:SR[23]=$SCR_GRP[1].$MCH_POS_X;
:SR[24]=$SCR_GRP[1].$MCH_POS_Y;
2027: L P[2027] 800cm/min CNT100 COORD PTH ;
:SR[23]=$SCR_GRP[1].$MCH_POS_X;
:SR[24]=$SCR_GRP[1].$MCH_POS_Y;
2028: L P[2028] 800cm/min CNT100 COORD PTH ;
:SR[23]=$SCR_GRP[1].$MCH_POS_X;
:SR[24]=$SCR_GRP[1].$MCH_POS_Y;
2029: L P[2029] 800cm/min CNT100 COORD PTH ;
:SR[23]=$SCR_GRP[1].$MCH_POS_X;
:SR[24]=$SCR_GRP[1].$MCH_POS_Y;
2030: L P[2030] 800cm/min CNT100 COORD PTH ;
:SR[23]=$SCR_GRP[1].$MCH_POS_X;
:SR[24]=$SCR_GRP[1].$MCH_POS_Y;
2031: L P[2031] 800cm/min CNT100 COORD PTH ;
:SR[23]=$SCR_GRP[1].$MCH_POS_X;
:SR[24]=$SCR_GRP[1].$MCH_POS_Y;
2032: L P[2032] 800cm/min CNT100 COORD PTH ;
:SR[23]=$SCR_GRP[1].$MCH_POS_X;
:SR[24]=$SCR_GRP[1].$MCH_POS_Y;
2033: L P[2033] 800cm/min CNT100 COORD PTH ;
:SR[23]=$SCR_GRP[1].$MCH_POS_X;
:SR[24]=$SCR_GRP[1].$MCH_POS_Y;
2034: L P[2034] 800cm/min CNT100 COORD PTH ;
:SR[23]=$SCR_GRP[1].$MCH_POS_X;
:SR[24]=$SCR_GRP[1].$MCH_POS_Y;
2035: L P[2035] 800cm/min CNT100 COORD PTH ;
:SR[23]=$SCR_GRP[1].$MCH_POS_X;
:SR[24]=$SCR_GRP[1].$MCH_POS_Y;
2036: L P[2036] 800cm/min CNT100 COORD PTH ;
:SR[23]=$SCR_GRP[1].$MCH_POS_X;
:SR[24]=$SCR_GRP[1].$MCH_POS_Y;
2037: L P[2037] 800cm/min CNT100 COORD PTH ;
:SR[23]=$SCR_GRP[1].$MCH_POS_X;
:SR[24]=$SCR_GRP[1].$MCH_POS_Y;
2038: L P[2038] 800cm/min CNT100 COORD PTH ;
:SR[23]=$SCR_GRP[1].$MCH_POS_X;
:SR[24]=$SCR_GRP[1].$MCH_POS_Y;
2039: L P[2039] 800cm/min CNT100 COORD PTH ;
:SR[23]=$SCR_GRP[1].$MCH_POS_X;
:SR[24]=$SCR_GRP[1].$MCH_POS_Y;
2040: L P[2040] 800cm/min CNT100 COORD PTH ;
:SR[23]=$SCR_GRP[1].$MCH_POS_X;
:SR[24]=$SCR_GRP[1].$MCH_POS_Y;
2041: L P[2041] 800cm/min CNT100 COORD PTH ;
:SR[23]=$SCR_GRP[1].$MCH_POS_X;
:SR[24]=$SCR_GRP[1].$MCH_POS_Y;
2042: L P[2042] 800cm/min CNT100 COORD PTH ;
:SR[23]=$SCR_GRP[1].$MCH_POS_X;
:SR[24]=$SCR_GRP[1].$MCH_POS_Y;
2043: L P[2043] 800cm/min CNT100 COORD PTH ;
:SR[23]=$SCR_GRP[1].$MCH_POS_X;
:SR[24]=$SCR_GRP[1].$MCH_POS_Y;
2044: L P[2044] 800cm/min CNT100 COORD PTH ;
:SR[23]=$SCR_GRP[1].$MCH_POS_X;
:SR[24]=$SCR_GRP[1].$MCH_POS_Y;
2045: L P[2045] 800cm/min CNT100 COORD PTH ;
:SR[23]=$SCR_GRP[1].$MCH_POS_X;
:SR[24]=$SCR_GRP[1].$MCH_POS_Y;
2046: L P[2046] 800cm/min CNT100 COORD PTH ;
:SR[23]=$SCR_GRP[1].$MCH_POS_X;
:SR[24]=$SCR_GRP[1].$MCH_POS_Y;
2047: L P[2047] 800cm/min CNT100 COORD PTH ;
:SR[23]=$SCR_GRP[1].$MCH_POS_X;
:SR[24]=$SCR_GRP[1].$MCH_POS_Y;
2048: L P[2048] 800cm/min CNT100 COORD PTH ;
:SR[23]=$SCR_GRP[1].$MCH_POS_X;
:SR[24]=$SCR_GRP[1].$MCH_POS_Y;
2049: L P[2049] 800cm/min CNT100 COORD PTH ;
:SR[23]=$SCR_GRP[1].$MCH_POS_X;
:SR[24]=$SCR_GRP[1].$MCH_POS_Y;
2050: L P[2050] 800cm/min CNT100 COORD PTH ;
:SR[23]=$SCR_GRP[1].$MCH_POS_X;
:SR[24]=$SCR_GRP[1].$MCH_POS_Y;
2051: L P[2051] 800cm/min CNT100 COORD PTH ;
:SR[23]=$SCR_GRP[1].$MCH_POS_X;
:SR[24]=$SCR_GRP[1].$MCH_POS_Y;
2052: L P[2052] 800cm/min CNT100 COORD PTH ;
:SR[23]=$SCR_GRP[1].$MCH_POS_X;
:SR[24]=$SCR_GRP[1].$MCH_POS_Y;
2053: L P[2053] 800cm/min CNT100 COORD PTH ;
:SR[23]=$SCR_GRP[1].$MCH_POS_X;
:SR[24]=$SCR_GRP[1].$MCH_POS_Y;
2054: L P[2054] 800cm/min CNT100 COORD PTH ;
:SR[23]=$SCR_GRP[1].$MCH_POS_X;
:SR[24]=$SCR_GRP[1].$MCH_POS_Y;
2055: L P[2055] 800cm/min CNT100 COORD PTH ;
:SR[23]=$SCR_GRP[1].$MCH_POS_X;
:SR[24]=$SCR_GRP[1].$MCH_POS_Y;
2056: L P[2056] 800cm/min CNT100 COORD PTH ;
:SR[23]=$SCR_GRP[1].$MCH_POS_X;
:SR[24]=$SCR_GRP[1].$MCH_POS_Y;
2057: L P[2057] 800cm/min CNT100 COORD PTH ;
:SR[23]=$SCR_GRP[1].$MCH_POS_X;
:SR[24]=$SCR_GRP[1].$MCH_POS_Y;
2058: L P[2058] 800cm/min CNT100 COORD PTH ;
:SR[23]=$SCR_GRP[1].$MCH_POS_X;
:SR[24]=$SCR_GRP[1].$MCH_POS_Y;
2059: L P[2059] 800cm/min CNT100 COORD PTH ;
:SR[23]=$SCR_GRP[1].$MCH_POS_X;
:SR[24]=$SCR_GRP[1].$MCH_POS_Y;
2060: L P[2060] 800cm/min CNT100 COORD PTH ;
:SR[23]=$SCR_GRP[1].$MCH_POS_X;
:SR[24]=$SCR_GRP[1].$MCH_POS_Y;
2061: L P[2061] 800cm/min CNT100 COORD PTH ;
:SR[23]=$SCR_GRP[1].$MCH_POS_X;
:SR[24]=$SCR_GRP[1].$MCH_POS_Y;
2062: L P[2062] 800cm/min CNT100 COORD PTH ;
:SR[23]=$SCR_GRP[1].$MCH_POS_X;
:SR[24]=$SCR_GRP[1].$MCH_POS_Y;
2063: L P[2063] 800cm/min CNT100 COORD PTH ;
:SR[23]=$SCR_GRP[1].$MCH_POS_X;
:SR[24]=$SCR_GRP[1].$MCH_POS_Y;
2064: L P[2064] 800cm/min CNT100 COORD PTH ;
:SR[23]=$SCR_GRP[1].$MCH_POS_X;
:SR[24]=$SCR_GRP[1].$MCH_POS_Y;
2065: L P[2065] 800cm/min CNT100 COORD PTH ;
:SR[23]=$SCR_GRP[1].$MCH_POS_X;
:SR[24]=$SCR_GRP[1].$MCH_POS_Y;
2066: L P[2066] 800cm/min CNT100 COORD PTH ;
:SR[23]=$SCR_GRP[1].$MCH_POS_X;
:SR[24]=$SCR_GRP[1].$MCH_POS_Y;
2067: L P[2067] 800cm/min CNT100 COORD PTH ;
:SR[23]=$SCR_GRP[1].$MCH_POS_X;
:SR[24]=$SCR_GRP[1].$MCH_POS_Y;
2068: L P[2068] 800cm/min CNT100 COORD PTH ;
:SR[23]=$SCR_GRP[1].$MCH_POS_X;
:SR[24]=$SCR_GRP[1].$MCH_POS_Y;
2069: L P[2069] 800cm/min CNT100 COORD PTH ;
:SR[23]=$SCR_GRP[1].$MCH_POS_X;
:SR[24]=$SCR_GRP[1].$MCH_POS_Y;
2070: L P[2070] 800cm/min CNT100 COORD PTH ;
:SR[23]=$SCR_GRP[1].$MCH_POS_X;
:SR[24]=$SCR_GRP[1].$MCH_POS_Y;
2071: L P[2071] 800cm/min CNT100 COORD PTH ;
:SR[23]=$SCR_GRP[1].$MCH_POS_X;
:SR[24]=$SCR_GRP[1].$MCH_POS_Y;
2072: L P[2072] 800cm/min CNT100 COORD PTH ;
:SR[23]=$SCR_GRP[1].$MCH_POS_X;
:SR[24]=$SCR_GRP[1].$MCH_POS_Y;
2073: L P[2073] 800cm/min CNT100 COORD PTH ;
:SR[23]=$SCR_GRP[1].$MCH_POS_X;
:SR[24]=$SCR_GRP[1].$MCH_POS_Y;
2074: L P[2074] 800cm/min CNT100 COORD PTH ;
:SR[23]=$SCR_GRP[1].$MCH_POS_X;
:SR[24]=$SCR_GRP[1].$MCH_POS_Y;
2075: L P[2075] 800cm/min CNT100 COORD PTH ;
:SR[23]=$SCR_GRP[1].$MCH_POS_X;
:SR[24]=$SCR_GRP[1].$MCH_POS_Y;
2076: L P[2076] 800cm/min CNT100 COORD PTH ;
:SR[23]=$SCR_GRP[1].$MCH_POS_X;
:SR[24]=$SCR_GRP[1].$MCH_POS_Y;
2077: L P[2077] 800cm/min CNT100 COORD PTH ;
:SR[23]=$SCR_GRP[1].$MCH_POS_X;
:SR[24]=$SCR_GRP[1].$MCH_POS_Y;
2078: L P[2078] 800cm/min CNT100 COORD PTH ;
:SR[23]=$SCR_GRP[1].$MCH_POS_X;
:SR[24]=$SCR_GRP[1].$MCH_POS_Y;
2079: L P[2079] 800cm/min CNT100 COORD PTH ;
:SR[23]=$SCR_GRP[1].$MCH_POS_X;
:SR[24]=$SCR_GRP[1].$MCH_POS_Y;
2080: L P[2080] 800cm/min CNT100 COORD PTH ;
:SR[23]=$SCR_GRP[1].$MCH_POS_X;
:SR[24]=$SCR_GRP[1].$MCH_POS_Y;
2081: L P[2081] 800cm/min CNT100 COORD PTH ;
:SR[23]=$SCR_GRP[1].$MCH_POS_X;
:SR[24]=$SCR_GRP[1].$MCH_POS_Y;
2082: L P[2082] 800cm/min CNT100 COORD PTH ;
:SR[23]=$SCR_GRP[1].$MCH_POS_X;
:SR[24]=$SCR_GRP[1].$MCH_POS_Y;
2083: L P[2083] 800cm/min CNT100 COORD PTH ;
:SR[23]=$SCR_GRP[1].$MCH_POS_X;
:SR[24]=$SCR_GRP[1].$MCH_POS_Y;
2084: L P[2084] 800cm/min CNT100 COORD PTH ;
:SR[23]=$SCR_GRP[1].$MCH_POS_X;
:SR[24]=$SCR_GRP[1].$MCH_POS_Y;
2085: L P[2085] 800cm/min CNT100 COORD PTH ;
:SR[23]=$SCR_GRP[1].$MCH_POS_X;
:SR[24]=$SCR_GRP[1].$MCH_POS_Y;
2086: L P[2086] 800cm/min CNT100 COORD PTH ;
:SR[23]=$SCR_GRP[1].$MCH_POS_X;
:SR[24]=$SCR_GRP[1].$MCH_POS_Y;
2087: L P[2087] 800cm/min CNT100 COORD PTH ;
:SR[23]=$SCR_GRP[1].$MCH_POS_X;
:SR[24]=$SCR_GRP[1].$MCH_POS_Y;
2088: L P[2088] 800cm/min CNT100 COORD PTH ;
:SR[23]=$SCR_GRP[1].$MCH_POS_X;
:SR[24]=$SCR_GRP[1].$MCH_POS_Y;
2089: L P[2089] 800cm/min CNT100 COORD PTH ;
:SR[23]=$SCR_GRP[1].$MCH_POS_X;
:SR[24]=$SCR_GRP[1].$MCH_POS_Y;
2090: L P[2090] 800cm/min CNT100 COORD PTH ;
:SR[23]=$SCR_GRP[1].$MCH_POS_X;
:SR[24]=$SCR_GRP[1].$MCH_POS_Y;
2091: L P[2091] 800cm/min CNT100 COORD PTH ;
:SR[23]=$SCR_GRP[1].$MCH_POS_X;
:SR[24]=$SCR_GRP[1].$MCH_POS_Y;
2092: L P[2092] 800cm/min CNT100 COORD PTH ;
:SR[23]=$SCR_GRP[1].$MCH_POS_X;
:SR[24]=$SCR_GRP[1].$MCH_POS_Y;
2093: L P[2093] 800cm/min CNT100 COORD PTH ;
:SR[23]=$SCR_GRP[1].$MCH_POS_X;
:SR[24]=$SCR_GRP[1].$MCH_POS_Y;
2094: L P[2094] 800cm/min CNT100 COORD PTH ;
:SR[23]=$SCR_GRP[1].$MCH_POS_X;
:SR[24]=$SCR_GRP[1].$MCH_POS_Y;
2095: L P[2095] 800cm/min CNT100 COORD PTH ;
:SR[23]=$SCR_GRP[1].$MCH_POS_X;
:SR[24]=$SCR_GRP[1].$MCH_POS_Y;
2096: L P[2096] 800cm/min CNT100 COORD PTH ;
:SR[23]=$SCR_GRP[1].$MCH_POS_X;
:SR[24]=$SCR_GRP[1].$MCH_POS_Y;
2097: L P[2097] 800cm/min CNT100 COORD PTH ;
:SR[23]=$SCR_GRP[1].$MCH_POS_X;
:SR[24]=$SCR_GRP[1].$MCH_POS_Y;
2098: L P[2098] 800cm/min CNT100 COORD PTH ;
:SR[23]=$SCR_GRP[1].$MCH_POS_X;
:SR[24]=$SCR_GRP[1].$MCH_POS_Y;
2099: L P[2099] 800cm/min CNT100 COORD PTH ;
:SR[23]=$SCR_GRP[1].$MCH_POS_X;
:SR[24]=$SCR_GRP[1].$MCH_POS_Y;
2100: L P[2100] 800cm/min CNT100 COORD PTH ;
:SR[23]=$SCR_GRP[1].$MCH_POS_X;
:SR[24]=$SCR_GRP[1].$MCH_POS_Y;
2101: L P[2101] 800cm/min CNT100 COORD PTH ;
:SR[23]=$SCR_GRP[1].$MCH_POS_X;
:SR[24]=$SCR_GRP[1].$MCH_POS_Y;
2102: L P[2102] 800cm/min CNT100 COORD PTH ;
:SR[23]=$SCR_GRP[1].$MCH_POS_X;
:SR[24]=$SCR_GRP[1].$MCH_POS_Y;
2103: L P[2103] 800cm/min CNT100 COORD PTH ;
:SR[23]=$SCR_GRP[1].$MCH_POS_X;
:SR[24]=$SCR_GRP[1].$MCH_POS_Y;
2104: L P[2104] 800cm/min CNT100 COORD PTH ;
:SR[23]=$SCR_GRP[1].$MCH_POS_X;
:SR[24]=$SCR_GRP[1].$MCH_POS_Y;
2105: L P[2105] 800cm/min CNT100 COORD PTH ;
:SR[23]=$SCR_GRP[1].$MCH_POS_X;
:SR[24]=$SCR_GRP[1].$MCH_POS_Y;
2106: L P[2106] 800cm/min CNT100 COORD PTH ;
:SR[23]=$SCR_GRP[1].$MCH_POS_X;
:SR[24]=$SCR_GRP[1].$MCH_POS_Y;
2107: L P[2107] 800cm/min CNT100 COORD PTH ;
:SR[23]=$SCR_GRP[1].$MCH_POS_X;
:SR[24]=$SCR_GRP[1].$MCH_POS_Y;
2108: L P[2108] 800cm/min CNT100 COORD PTH ;
:SR[23]=$SCR_GRP[1].$MCH_POS_X;
:SR[24]=$SCR_GRP[1].$MCH_POS_Y;
2109: L P[2109] 800cm/min CNT100 COORD PTH ;
:SR[23]=$SCR_GRP[1].$MCH_POS_X;
:SR[24]=$SCR_GRP[1].$MCH_POS_Y;
2110: L P[2110] 800cm/min CNT100 COORD PTH ;
:SR[23]=$SCR_GRP[1].$MCH_POS_X;
:SR[24]=$SCR_GRP[1].$MCH_POS_Y;
2111: L P[2111] 800cm/min CNT100 COORD PTH ;
:SR[23]=$SCR_GRP[1].$MCH_POS_X;
:SR[24]=$SCR_GRP[1].$MCH_POS_Y;
2112: L P[2112] 800cm/min CNT100 COORD PTH ;
:SR[23]=$SCR_GRP[1].$MCH_POS_X;
:SR[24]=$SCR_GRP[1].$MCH_POS_Y;
2113: L P[2113] 800cm/min CNT100 COORD PTH ;
:SR[23]=$SCR_GRP[1].$MCH_POS_X;
:SR[24]=$SCR_GRP[1].$MCH_POS_Y;
2114: L P[2114] 800cm/min CNT100 COORD PTH ;
:SR[23]=$SCR_GRP[1].$MCH_POS_X;
:SR[24]=$SCR_GRP[1].$MCH_POS_Y;
2115: L P[2115] 800cm/min CNT100 COORD PTH ;
:SR[23]=$SCR_GRP[1].$MCH_POS_X;
:SR[24]=$SCR_GRP[1].$MCH_POS_Y;
2116: L P[2116] 800cm/min CNT100 COORD PTH ;
:SR[23]=$SCR_GRP[1].$MCH_POS_X;
:SR[24]=$SCR_GRP[1].$MCH_POS_Y;
2117: L P[2117] 800cm/min CNT100 COORD PTH ;
:SR[23]=$SCR_GRP[1].$MCH_POS_X;
:SR[24]=$SCR_GRP[1].$MCH_POS_Y;
2118: L P[2118] 800cm/min CNT100 COORD PTH ;
:SR[23]=$SCR_GRP[1].$MCH_POS_X;
:SR[24]=$SCR_GRP[1].$MCH_POS_Y;
2119: L P[2119] 800cm/min CNT100 COORD PTH ;
:SR[23]=$SCR_GRP[1].$MCH_POS_X;
:SR[24]=$SCR_GRP[1].$MCH_POS_Y;
2120: L P[2120] 800cm/min CNT100 COORD PTH ;
:SR[23]=$SCR_GRP[1].$MCH_POS_X;
:SR[24]=$SCR_GRP[1].$MCH_POS_Y;
2121: L P[2121] 800cm/min CNT100 COORD PTH ;
:SR[23]=$SCR_GRP[1].$MCH_POS_X;
:SR[24]=$SCR_GRP[1].$MCH_POS_Y;
2122: L P[2122] 800cm/min CNT100 COORD PTH ;
:SR[23]=$SCR_GRP[1].$MCH_POS_X;
:SR[24]=$SCR_GRP[1].$MCH_POS_Y;
2123: L P[2123] 800cm/min CNT100 COORD PTH ;
:SR[23]=$SCR_GRP[1].$MCH_POS_X;
:SR[24]=$SCR_GRP[1].$MCH_POS_Y;
2124: L P[2124] 800cm/min CNT100 COORD PTH ;
:SR[23]=$SCR_GRP[1].$MCH_POS_X;
:SR[24]=$SCR_GRP[1].$MCH_POS_Y;
2125: L P[2125] 800cm/min CNT100 COORD PTH ;
:SR[23]=$SCR_GRP[1].$MCH_POS_X;
:SR[24]=$SCR_GRP[1].$MCH_POS_Y;
2126: L P[2126] 800cm/min CNT100 COORD PTH ;
:SR[23]=$SCR_GRP[1].$MCH_POS_X;
:SR[24]=$SCR_GRP[1].$MCH_POS_Y;
2127: L P[2127] 800cm/min CNT100 COORD PTH ;
:SR[23]=$SCR_GRP[1].$MCH_POS_X;
:SR[24]=$SCR_GRP[1].$MCH_POS_Y;
2128: L P[2128] 800cm/min CNT100 COORD PTH ;
:SR[23]=$SCR_GRP[1].$MCH_POS_X;
:SR[24]=$SCR_GRP[1].$MCH_POS_Y;
2129: L P[2129] 800cm/min CNT100 COORD PTH ;
:SR[23]=$SCR_GRP[1].$MCH_POS_X;
:SR[24]=$SCR_GRP[1].$MCH_POS_Y;
2130: L P[2130] 800cm/min CNT100 COORD PTH ;
:SR[23]=$SCR_GRP[1].$MCH_POS_X;
:SR[24]=$SCR_GRP[1].$MCH_POS_Y;
2131: L P[2131] 800cm/min CNT100 COORD PTH ;
:SR[23]=$SCR_GRP[1].$MCH_POS_X;
:SR[24]=$SCR_GRP[1].$MCH_POS_Y;
2132: L P[2132] 800cm/min CNT100 COORD PTH ;
:SR[23]=$SCR_GRP[1].$MCH_POS_X;
:SR[24]=$SCR_GRP[1].$MCH_POS_Y;
2133: L P[2133] 800cm/min CNT100 COORD PTH ;
:SR[23]=$SCR_GRP[1].$MCH_POS_X;
:SR[24]=$SCR_GRP[1].$MCH_POS_Y;
2134: L P[2134] 800cm/min CNT100 COORD PTH ;
:SR[23]=$SCR_GRP[1].$MCH_POS_X;
:SR[24]=$SCR_GRP[1].$MCH_POS_Y;
2135: L P[2135] 800cm/min CNT100 COORD PTH ;
:SR[23]=$SCR_GRP[1].$MCH_POS_X;
:SR[24]=$SCR_GRP[1].$MCH_POS_Y;
2136: L P[2136] 800cm/min CNT100 COORD PTH ;
:SR[23]=$SCR_GRP[1].$MCH_POS_X;
:SR[24]=$SCR_GRP[1].$MCH_POS_Y;
2137: L P[2137] 800cm/min CNT100 COORD PTH ;
:SR[23]=$SCR_GRP[1].$MCH_POS_X;
:SR[24]=$SCR_GRP[1].$MCH_POS_Y;
2138: L P[2138] 800cm/min CNT100 COORD PTH ;
:SR[23]=$SCR_GRP[1].$MCH_POS_X;
:SR[24]=$SCR_GRP[1].$MCH_POS_Y;
2139: L P[2139] 800cm/min CNT100 COORD PTH ;
:SR[23]=$SCR_GRP[1].$MCH_POS_X;
:SR[24]=$SCR_GRP[1].$MCH_POS_Y;
2140: L P[2140] 800cm/min CNT100 COORD PTH ;
:SR[23]=$SCR_GRP[1].$MCH_POS_X;
:SR[24]=$SCR_GRP[1].$MCH_POS_Y;
2141: L P[2141] 800cm/min CNT100 COORD PTH ;
:SR[23]=$SCR_GRP[1].$MCH_POS_X;
:SR[24]=$SCR_GRP[1].$MCH_POS_Y;
2142: L P[2142] 800cm/min CNT100 COORD PTH ;
:SR[23]=$SCR_GRP[1].$MCH_POS_X;
:SR[24]=$SCR_GRP[1].$MCH_POS_Y;
2143: L P[2143] 800cm/min CNT100 COORD PTH ;
:SR[23]=$SCR_GRP[1].$MCH_POS_X;
:SR[24]=$SCR_GRP[1].$MCH_POS_Y;
2144: L P[2144] 800cm/min CNT100 COORD PTH ;
:SR[23]=$SCR_GRP[1].$MCH_POS_X;
:SR[24]=$SCR_GRP[1].$MCH_POS_Y;
2145: L P[2145] 800cm/min CNT100 COORD PTH ;
:SR[23]=$SCR_GRP[1].$MCH_POS_X;
:SR[24]=$SCR_GRP[1].$MCH_POS_Y;
2146: L P[2146] 800cm/min CNT100 COORD PTH ;
:SR[23]=$SCR_GRP[1].$MCH_POS_X;
:SR[24]=$SCR_GRP[1].$MCH_POS_Y;
2147: L P[2147] 800cm/min CNT100 COORD PTH ;
:SR[23]=$SCR_GRP[1].$MCH_POS_X;
:SR[24]=$SCR_GRP[1].$MCH_POS_Y;
2148: L P[2148] 800cm/min CNT100 COORD PTH ;
:SR[23]=$SCR_GRP[1].$MCH_POS_X;
:SR[24]=$SCR_GRP[1].$MCH_POS_Y;
2149: L P[2149] 800cm/min CNT100 COORD PTH ;
:SR[23]=$SCR_GRP[1].$MCH_POS_X;
:SR[24]=$SCR_GRP[1].$MCH_POS_Y;
2150: L P[2150] 800cm/min CNT100 COORD PTH ;
:SR[23]=$SCR_GRP[1].$MCH_POS_X;
:SR[24]=$SCR_GRP[1].$MCH_POS_Y;
2151: L P[2151] 800cm/min CNT100 COORD PTH ;
:SR[23]=$SCR_GRP[1].$MCH_POS_X;
:SR[24]=$SCR_GRP[1].$MCH_POS_Y;
2152: L P[2152] 800cm/min CNT100 COORD PTH ;
:SR[23]=$SCR_GRP[1].$MCH_POS_X;
:SR[24]=$SCR_GRP[1].$MCH_POS_Y;
2153: L P[2153] 800cm/min CNT100 COORD PTH ;
:SR[23]=$SCR_GRP[1].$MCH_POS_X;
:SR[24]=$SCR_GRP[1].$MCH_POS_Y;
2154: L P[2154] 800cm/min CNT100 COORD PTH ;
:SR[23]=$SCR_GRP[1].$MCH_POS_X;
:SR[24]=$SCR_GRP[1].$MCH_POS_Y;
2155: L P[2155] 800cm/min CNT100 COORD PTH ;
:SR[23]=$SCR_GRP[1].$MCH_POS_X;
:SR[24]=$SCR_GRP[1].$MCH_POS_Y;
2156: L P[2156] 800cm/min CNT100 COORD PTH ;
:SR[23]=$SCR_GRP[1].$MCH_POS_X;
:SR[24]=$SCR_GRP[1].$MCH_POS_Y;
2157: L P[2157] 800cm/min CNT100 COORD PTH ;
:SR[23]=$SCR_GRP[1].$MCH_POS_X;
:SR[24]=$SCR_GRP[1].$MCH_POS_Y;
2158: L P[2158] 800cm/min CNT100 COORD PTH ;
:SR[23]=$SCR_GRP[1].$MCH_POS_X;
:SR[24]=$SCR_GRP[1].$MCH_POS_Y;
2159: L P[2159] 800cm/min CNT100 COORD PTH ;
:SR[23]=$SCR_GRP[1].$MCH_POS_X;
:SR[24]=$SCR_GRP[1].$MCH_POS_Y;
2160: L P[2160] 800cm/min CNT100 COORD PTH ;
:SR[23]=$SCR_GRP[1].$MCH_POS_X;
:SR[24]=$SCR_GRP[1].$MCH_POS_Y;
2161: L P[2161] 800cm/min CNT100 COORD PTH ;
:SR[23]=$SCR_GRP[1].$MCH_POS_X;
:SR[24]=$SCR_GRP[1].$MCH_POS_Y;
2162: L P[2162] 800cm/min CNT100 COORD PTH ;
:SR[23]=$SCR_GRP[1].$MCH_POS_X;
:SR[24]=$SCR_GRP[1].$MCH_POS_Y;
2163: L P[2163] 800cm/min CNT100 COORD PTH ;
:SR[23]=$SCR_GRP[1].$MCH_POS_X;
:SR[24]=$SCR_GRP[1].$MCH_POS_Y;
2164: L P[2164] 800cm/min CNT100 COORD PTH ;
:SR[23]=$SCR_GRP[1].$MCH_POS_X;
:SR[24]=$SCR_GRP[1].$MCH_POS_Y;
2165: L P[2165] 800cm/min CNT100 COORD PTH ;
:SR[23]=$SCR_GRP[1].$MCH_POS_X;
:SR[24]=$SCR_GRP[1].$MCH_POS_Y;
2166: L P[2166] 800cm/min CNT100 COORD PTH ;
:SR[23]=$SCR_GRP[1].$MCH_POS_X;
:SR[24]=$SCR_GRP[1].$MCH_POS_Y;
2167: L P[2167] 800cm/min CNT100 COORD PTH ;
:SR[23]=$SCR_GRP[1].$MCH_POS_X;
:SR[24]=$SCR_GRP[1].$MCH_POS_Y;
2168: L P[2168] 800cm/min CNT100 COORD PTH ;
:SR[23]=$SCR_GRP[1].$MCH_POS_X;
:SR[24]=$SCR_GRP[1].$MCH_POS_Y;
2169: L P[2169] 800cm/min CNT100 COORD PTH ;
:SR[23]=$SCR_GRP[1].$MCH_POS_X;
:SR[24]=$SCR_GRP[1].$MCH_POS_Y;
2170: L P[2170] 800cm/min CNT100 COORD PTH ;
:SR[23]=$SCR_GRP[1].$MCH_POS_X;
:SR[24]=$SCR_GRP[1].$MCH_POS_Y;
2171: L P[2171] 800cm/min CNT100 COORD PTH ;
:SR[23]=$SCR_GRP[1].$MCH_POS_X;
:SR[24]=$SCR_GRP[1].$MCH_POS_Y;
2172: L P[2172] 800cm/min CNT100 COORD PTH ;
:SR[23]=$SCR_GRP[1].$MCH_POS_X;
:SR[24]=$SCR_GRP[1].$MCH_POS_Y;
2173: L P[2173] 800cm/min CNT100 COORD PTH ;
:SR[23]=$SCR_GRP[1].$MCH_POS_X;
:SR[24]=$SCR_GRP[1].$MCH_POS_Y;
2174: L P[2174] 800cm/min CNT100 COORD PTH ;
:SR[23]=$SCR_GRP[1].$MCH_POS_X;
:SR[24]=$SCR_GRP[1].$MCH_POS_Y;
2175: L P[2175] 800cm/min CNT100 COORD PTH ;
:SR[23]=$SCR_GRP[1].$MCH_POS_X;
:SR[24]=$SCR_GRP[1].$MCH_POS_Y;
2176: L P[2176] 800cm/min CNT100 COORD PTH ;
:SR[23]=$SCR_GRP[1].$MCH_POS_X;
:SR[24]=$SCR_GRP[1].$MCH_POS_Y;
2177: L P[2177] 800cm/min CNT100 COORD PTH ;
:SR[23]=$SCR_GRP[1].$MCH_POS_X;
:SR[24]=$SCR_GRP[1].$MCH_POS_Y;
2178: L P[2178] 800cm/min CNT100 COORD PTH ;
:SR[23]=$SCR_GRP[1].$MCH_POS_X;
:SR[24]=$SCR_GRP[1].$MCH_POS_Y;
2179: L P[2179] 800cm/min CNT100 COORD PTH ;
:SR[23]=$SCR_GRP[1].$MCH_POS_X;
:SR[24]=$SCR_GRP[1].$MCH_POS_Y;
2180: L P[2180] 800cm/min CNT100 COORD PTH ;
:SR[23]=$SCR_GRP[1].$MCH_POS_X;
:SR[24]=$SCR_GRP[1].$MCH_POS_Y;
2181: L P[2181] 800cm/min CNT100 COORD PTH ;
:SR[23]=$SCR_GRP[1].$MCH_POS_X;
:SR[24]=$SCR_GRP[1].$MCH_POS_Y;
2182: L P[2182] 800cm/min CNT100 COORD PTH ;
:SR[23]=$SCR_GRP[1].$MCH_POS_X;
:SR[24]=$SCR_GRP[1].$MCH_POS_Y;
2183: L P[2183] 800cm/min CNT100 COORD PTH ;
:SR[23]=$SCR_GRP[1].$MCH_POS_X;
:SR[24]=$SCR_GRP[1].$MCH_POS_Y;
2184: L P[2184] 800cm/min CNT100 COORD PTH ;
:SR[23]=$SCR_GRP[1].$MCH_POS_X;
:SR[24]=$SCR_GRP[1].$MCH_POS_Y;
2185: L P[2185] 800cm/min CNT100 COORD PTH ;
:SR[23]=$SCR_GRP[1].$MCH_POS_X;
:SR[24]=$SCR_GRP[1].$MCH_POS_Y;
2186: L P[2186] 800cm/min CNT100 COORD PTH ;
:SR[23]=$SCR_GRP[1].$MCH_POS_X;
:SR[24]=$SCR_GRP[1].$MCH_POS_Y;
2187: L P[2187] 800cm/min CNT100 COORD PTH ;
:SR[23]=$SCR_GRP[1].$MCH_POS_X;
:SR[24]=$SCR_GRP[1].$MCH_POS_Y;
2188: L P[2188] 800cm/min CNT100 COORD PTH ;
:SR[23]=$SCR_GRP[1].$MCH_POS_X;
:SR[24]=$SCR_GRP[1].$MCH_POS_Y;
2189: L P[2189] 800cm/min CNT100 COORD PTH ;
:SR[23]=$SCR_GRP[1].$MCH_POS_X;
:SR[24]=$SCR_GRP[1].$MCH_POS_Y;
2190: L P[2190] 800cm/min CNT100 COORD PTH ;
:SR[23]=$SCR_GRP[1].$MCH_POS_X;
:SR[24]=$SCR_GRP[1].$MCH_POS_Y;
2191: L P[2191] 800cm/min CNT100 COORD PTH ;
:SR[23]=$SCR_GRP[1].$MCH_POS_X;
:SR[24]=$SCR_GRP[1].$MCH_POS_Y;
2192: L P[2192] 800cm/min CNT100 COORD PTH ;
:SR[23]=$SCR_GRP[1].$MCH_POS_X;
:SR[24]=$SCR_GRP[1].$MCH_POS_Y;
2193: L P[2193] 800cm/min CNT100 COORD PTH ;
:SR[23]=$SCR_GRP[1].$MCH_POS_X;
:SR[24]=$SCR_GRP[1].$MCH_POS_Y;
2194: L P[2194] 800cm/min CNT100 COORD PTH ;
:SR[23]=$SCR_GRP[1].$MCH_POS_X;
:SR[24]=$SCR_GRP[1].$MCH_POS_Y;
2195: L P[2195] 800cm/min CNT100 COORD PTH ;
:SR[23]=$SCR_GRP[1].$MCH_POS_X;
:SR[24]=$SCR_GRP[1].$MCH_POS_Y;
2196: L P[2196] 800cm/min CNT100 COORD PTH ;
:SR[23]=$SCR_GRP[1].$MCH_POS_X;
:SR[24]=$SCR_GRP[1].$MCH_POS_Y;
2197: L P[2197] 800cm/min CNT100 COORD PTH ;
:SR[23]=$SCR_GRP[1].$MCH_POS_X;
:SR[24]=$SCR_GRP[1].$MCH_POS_Y;
2198: L P[2198] 800cm/min CNT100 COORD PTH ;
:SR[23]=$SCR_GRP[1].$MCH_POS_X;
:SR[24]=$SCR_GRP[1].$MCH_POS_Y;
2199: L P[2199] 800cm/min CNT100 COORD PTH ;
:SR[23]=$SCR_GRP[1].$MCH_POS_X;
:SR[24]=$SCR_GRP[1].$MCH_POS_Y;
2200: L P[2200] 800cm/min CNT100 COORD PTH ;
:SR[23]=$SCR_GRP[1].$MCH_POS_X;
:SR[24]=$SCR_GRP[1].$MCH_POS_Y;
2201: L P[2201] 800cm/min CNT100 COORD PTH ;
:SR[23]=$SCR_GRP[1].$MCH_POS_X;
:SR[24]=$SCR_GRP[1].$MCH_POS_Y;
2202: L P[2202] 800cm/min CNT100 COORD PTH ;
:SR[23]=$SCR_GRP[1].$MCH_POS_X;
:SR[24]=$SCR_GRP[1].$MCH_POS_Y;
2203: L P[2203] 800cm/min CNT100 COORD PTH ;
:SR[23]=$SCR_GRP[1].$MCH_POS_X;
:SR[24]=$SCR_GRP[1].$MCH_POS_Y;
2204: L P[2204] 800cm/min CNT100 COORD PTH ;
:SR[23]=$SCR_GRP[1].$MCH_POS_X;
:SR[24]=$SCR_GRP[1].$MCH_POS_Y;
2205: L P[2205] 800cm/min CNT100 COORD PTH ;
:SR[23]=$SCR_GRP[1].$MCH_POS_X;
:SR[24]=$SCR_GRP[1].$MCH_POS_Y;
2206: L P[2206] 800cm/min CNT100 COORD PTH ;
:SR[23]=$SCR_GRP[1].$MCH_POS_X;
:SR[24]=$SCR_GRP[1].$MCH_POS_Y;
2207: L P[2207] 800cm/min CNT100 COORD PTH ;
:SR[23]=$SCR_GRP[1].$MCH_POS_X;
:SR[24]=$SCR_GRP[1].$MCH_POS_Y;
2208: L P[2208] 800cm/min CNT100 COORD PTH ;
:SR[23]=$SCR_GRP[1].$MCH_POS_X;
:SR[24]=$SCR_GRP[1].$MCH_POS_Y;
2209: L P[2209] 800cm/min CNT100 COORD PTH ;
:SR[23]=$SCR_GRP[1].$MCH_POS_X;
:SR[24]=$SCR_GRP[1].$MCH_POS_Y;
2210: L P[2210] 800cm/min CNT100 COORD PTH ;
:SR[23]=$SCR_GRP[1].$MCH_POS_X;
:SR[24]=$SCR_GRP[1].$MCH_POS_Y;
2211: L P[2211] 800cm/min CNT100 COORD PTH ;
:SR[23]=$SCR_GRP[1].$MCH_POS_X;
:SR[24]=$SCR_GRP[1].$MCH_POS_Y;
2212: L P[2212] 800cm/min CNT100 COORD PTH ;
:SR[23]=$SCR_GRP[1].$MCH_POS_X;
:SR[24]=$SCR_GRP[1].$MCH_POS_Y;
2213: L P[2213] 800cm/min CNT100 COORD PTH ;
:SR[23]=$SCR_GRP[1].$MCH_POS_X;
:SR[24]=$SCR_GRP[1].$MCH_POS_Y;
2214: L P[2214] 800cm/min CNT100 COORD PTH ;
:SR[23]=$SCR_GRP[1].$MCH_POS_X;
:SR[24]=$SCR_GRP[1].$MCH_POS_Y;
2215: L P[2215] 800cm/min CNT100 COORD PTH ;
:SR[23]=$SCR_GRP[1].$MCH_POS_X;
:SR[24]=$SCR_GRP[1].$MCH_POS_Y;
2216: L P[2216] 800cm/min CNT100 COORD PTH ;
:SR[23]=$SCR_GRP[1].$MCH_POS_X;
:SR[24]=$SCR_GRP[1].$MCH_POS_Y;
2217: L P[2217] 800cm/min CNT100 COORD PTH ;
:SR[23]=$SCR_GRP[1].$MCH_POS_X;
:SR[24]=$SCR_GRP[1].$MCH_POS_Y;
2218: L P[2218] 800cm/min CNT100 COORD PTH ;
:SR[23]=$SCR_GRP[1].$MCH_POS_X;
:SR[24]=$SCR_GRP[1].$MCH_POS_Y;
2219: L P[2219] 800cm/min CNT100 COORD PTH ;
:SR[23]=$SCR_GRP[1].$MCH_POS_X;
:SR[24]=$SCR_GRP[1].$MCH_POS_Y;
2220: L P[2220] 800cm/min CNT100 COORD PTH ;
:SR[23]=$SCR_GRP[1].$MCH_POS_X;
:SR[24]=$SCR_GRP[1].$MCH_POS_Y;
2221: L P[2221] 800cm/min CNT100 COORD PTH ;
:SR[23]=$SCR_GRP[1].$MCH_POS_X;
:SR[24]=$SCR_GRP[1].$MCH_POS_Y;
2222: L P[2222] 800cm/min CNT100 COORD PTH ;
:SR[23]=$SCR_GRP[1].$MCH_POS_X;
:SR[24]=$SCR_GRP[1].$MCH_POS_Y;
2223: L P[2223] 800cm/min CNT100 COORD PTH ;
:SR[23]=$SCR_GRP[1].$MCH_POS_X;
:SR[24]=$SCR_GRP[1].$MCH_POS_Y;
2224: L P[2224] 800cm/min CNT100 COORD PTH ;
:SR[23]=$SCR_GRP[1].$MCH_POS_X;
:SR[24]=$SCR_GRP[1].$MCH_POS_Y;
2225: L P[2225] 800cm/min CNT100 COORD PTH ;
:SR[23]=$SCR_GRP[1].$MCH_POS_X;
:SR[24]=$SCR_GRP[1].$MCH_POS_Y;
2226: L P[2226] 800cm/min CNT100 COORD PTH ;
:SR[23]=$SCR_GRP[1].$MCH_POS_X;
:SR[24]=$SCR_GRP[1].$MCH_POS_Y;
2227: L P[2227] 800cm/min CNT100 COORD PTH ;
:SR[23]=$SCR_GRP[1].$MCH_POS_X;
:SR[24]=$SCR_GRP[1].$MCH_POS_Y;
2228: L P[2228] 800cm/min CNT100 COORD PTH ;
:SR[23]=$SCR_GRP[1].$MCH_POS_X;
:SR[24]=$SCR_GRP[1].$MCH_POS_Y;
2229: L P[2229] 800cm/min CNT100 COORD PTH ;
:SR[23]=$SCR_GRP[1].$MCH_POS_X;
:SR[24]=$SCR_GRP[1].$MCH_POS_Y;
2230: L P[2230] 800cm/min CNT100 COORD PTH ;
:SR[23]=$SCR_GRP[1].$MCH_POS_X;
:SR[24]=$SCR_GRP[1].$MCH_POS_Y;
2231: L P[2231] 800cm/min CNT100 COORD PTH ;
:SR[23]=$SCR_GRP[1].$MCH_POS_X;
:SR[24]=$SCR_GRP[1].$MCH_POS_Y;
2232: L P[2232] 800cm/min CNT100 COORD PTH ;
:SR[23]=$SCR_GRP[1].$MCH_POS_X;
:SR[24]=$SCR_GRP[1].$MCH_POS_Y;
2233: L P[2233] 800cm/min CNT100 COORD PTH ;
:SR[23]=$SCR_GRP[1].$MCH_POS_X;
:SR[24]=$SCR_GRP[1].$MCH_POS_Y;
2234: L P[2234] 800cm/min CNT100 COORD PTH ;
:SR[23]=$SCR_GRP[1].$MCH_POS_X;
:SR[24]=$SCR_GRP[1].$MCH_POS_Y;
2235: L P[2235] 800cm/min CNT100 COORD PTH ;
:SR[23]=$SCR_GRP[1].$MCH_POS_X;
:SR[24]=$SCR_GRP[1].$MCH_POS_Y;
2236: L P[2236] 800cm/min CNT100 COORD PTH ;
:SR[23]=$SCR_GRP[1].$MCH_POS_X;
:SR[24]=$SCR_GRP[1].$MCH_POS_Y;
2237: L P[2237] 800cm/min CNT100 COORD PTH ;
:SR[23]=$SCR_GRP[1].$MCH_POS_X;
:SR[24]=$SCR_GRP[1].$MCH_POS_Y;
2238: L P[2238] 800cm/min CNT100 COORD PTH ;
:SR[23]=$SCR_GRP[1].$MCH_POS_X;
:SR[24]=$SCR_GRP[1].$MCH_POS_Y;
2239: L P[2239] 800cm/min CNT100 COORD PTH ;
:SR[23]=$SCR_GRP[1].$MCH_POS_X;
:SR[24]=$SCR_GRP[1].$MCH_POS_Y;
2240: L P[2240] 800cm/min CNT100 COORD PTH ;
:SR[23]=$SCR_GRP[1].$MCH_POS_X;
:SR[24]=$SCR_GRP[1].$MCH_POS_Y;
2241: L P[2241] 800cm/min CNT100 COORD PTH ;
:SR[23]=$SCR_GRP[1].$MCH_POS_X;
:SR[24]=$SCR_GRP[1].$MCH_POS_Y;
2242: L P[2242] 800cm/min CNT100 COORD PTH ;
:SR[23]=$SCR_GRP[1].$MCH_POS_X;
:SR[24]=$SCR_GRP[1].$MCH_POS_Y;
2243: L P[2243] 800cm/min CNT100 COORD PTH ;
:SR[23]=$SCR_GRP[1].$MCH_POS_X;
:SR[24]=$SCR_GRP[1].$MCH_POS_Y;
2244: L P[2244] 800cm/min CNT100 COORD PTH ;
:SR[23]=$SCR_GRP[1].$MCH_POS_X;
:SR[24]=$SCR_GRP[1].$MCH_POS_Y;
2245: L P[2245] 800cm/min CNT100 COORD PTH ;
:SR[23]=$SCR_GRP[1].$MCH_POS_X;
:SR[24]=$SCR_GRP[1].$MCH_POS_Y;
2246: L P[2246] 800cm/min CNT100 COORD PTH ;
:SR[23]=$SCR_GRP[1].$MCH_POS_X;
:SR[24]=$SCR_GRP[1].$MCH_POS_Y;
2247: L P[2247] 800cm/min CNT100 COORD PTH ;
:SR[23]=$SCR_GRP[1].$MCH_POS_X;
:SR[24]=$SCR_GRP[1].$MCH_POS_Y;
2248: L P[2248] 800cm/min CNT100 COORD PTH ;
:SR[23]=$SCR_GRP[1].$MCH_POS_X;
:SR[24]=$SCR_GRP[1].$MCH_POS_Y;
2249: L P[2249] 800cm/min CNT100 COORD PTH ;
:SR[23]=$SCR_GRP[1].$MCH_POS_X;
:SR[24]=$SCR_GRP[1].$MCH_POS_Y;
2250: L P[2250] 800cm/min CNT100 COORD PTH ;
:SR[23]=$SCR_GRP[1].$MCH_POS_X;
:SR[24]=$SCR_GRP[1].$MCH_POS_Y;
2251: L P[2251] 800cm/min CNT100 COORD PTH ;
:SR[23]=$SCR_GRP[1].$MCH_POS_X;
:SR[24]=$SCR_GRP[1].$MCH_POS_Y;
2252: L P[2252] 800cm/min CNT100 COORD PTH ;
:SR[23]=$SCR_GRP[1].$MCH_POS_X;
:SR[24]=$SCR_GRP[1].$MCH_POS_Y;
2253: L P[2253] 800cm/min CNT100 COORD PTH ;
:SR[23]=$SCR_GRP[1].$MCH_POS_X;
:SR[24]=$SCR_GRP[1].$MCH_POS_Y;
2254: L P[2254] 800cm/min CNT100 COORD PTH ;
:SR[23]=$SCR_GRP[1].$MCH_POS_X;
:SR[24]=$SCR_GRP[1].$MCH_POS_Y;
2255: L P[2255] 800cm/min CNT100 COORD PTH ;
:SR[23]=$SCR_GRP[1].$MCH_POS_X;
:SR[24]=$SCR_GRP[1].$MCH_POS_Y;
2256: L P[2256] 800cm/min CNT100 COORD PTH ;
:SR[23]=$SCR_GRP[1].$MCH_POS_X;
:SR[24]=$SCR_GRP[1].$MCH_POS_Y;
2257: L P[2257] 800cm/min CNT100 COORD PTH ;
:SR[23]=$SCR_GRP[1].$MCH_POS_X;
:SR[24]=$SCR_GRP[1].$MCH_POS_Y;
2258: L P[2258] 800cm/min CNT100 COORD PTH ;
:SR[23]=$SCR_GRP[1].$MCH_POS_X;
:SR[24]=$SCR_GRP[1].$MCH_POS_Y;
2259: L P[2259] 800cm/min CNT100 COORD PTH ;
:SR[23]=$SCR_GRP[1].$MCH_POS_X;
:SR[24]=$SCR_GRP[1].$MCH_POS_Y;
2260: L P[2260] 800cm/min CNT100 COORD PTH ;
:SR[23]=$SCR_GRP[1].$MCH_POS_X;
:SR[24]=$SCR_GRP[1].$MCH_POS_Y;
2261: L P[2261] 800cm/min CNT100 COORD PTH ;
:SR[23]=$SCR_GRP[1].$MCH_POS_X;
:SR[24]=$SCR_GRP[1].$MCH_POS_Y;
2262: L P[2262] 800cm/min CNT100 COORD ;
:SR[23]=$SCR_GRP[1].$MCH_POS_X;
:SR[24]=$SCR_GRP[1].$MCH_POS_Y;
2263: L P[2263] 800cm/min CNT100 COORD PTH ;
:SR[23]=$SCR_GRP[1].$MCH_POS_X;
:SR[24]=$SCR_GRP[1].$MCH_POS_Y;
2264: L P[2264] 800cm/min CNT100 COORD PTH ;
:SR[23]=$SCR_GRP[1].$MCH_POS_X;
:SR[24]=$SCR_GRP[1].$MCH_POS_Y;
2265: L P[2265] 800cm/min CNT100 COORD PTH ;
:SR[23]=$SCR_GRP[1].$MCH_POS_X;
:SR[24]=$SCR_GRP[1].$MCH_POS_Y;
2266: L P[2266] 800cm/min CNT100 COORD PTH ;
:SR[23]=$SCR_GRP[1].$MCH_POS_X;
:SR[24]=$SCR_GRP[1].$MCH_POS_Y;
2267: L P[2267] 800cm/min CNT100 COORD PTH ;
:SR[23]=$SCR_GRP[1].$MCH_POS_X;
:SR[24]=$SCR_GRP[1].$MCH_POS_Y;
2268: L P[2268] 800cm/min CNT100 COORD PTH ;
:SR[23]=$SCR_GRP[1].$MCH_POS_X;
:SR[24]=$SCR_GRP[1].$MCH_POS_Y;
2269: L P[2269] 800cm/min CNT100 COORD PTH ;
:SR[23]=$SCR_GRP[1].$MCH_POS_X;
:SR[24]=$SCR_GRP[1].$MCH_POS_Y;
2270: L P[2270] 800cm/min CNT100 COORD PTH ;
:SR[23]=$SCR_GRP[1].$MCH_POS_X;
:SR[24]=$SCR_GRP[1].$MCH_POS_Y;
2271: L P[2271] 800cm/min CNT100 COORD PTH ;
:SR[23]=$SCR_GRP[1].$MCH_POS_X;
:SR[24]=$SCR_GRP[1].$MCH_POS_Y;
2272: L P[2272] 800cm/min CNT100 COORD PTH ;
:SR[23]=$SCR_GRP[1].$MCH_POS_X;
:SR[24]=$SCR_GRP[1].$MCH_POS_Y;
2273: L P[2273] 800cm/min CNT100 COORD PTH ;
:SR[23]=$SCR_GRP[1].$MCH_POS_X;
:SR[24]=$SCR_GRP[1].$MCH_POS_Y;
2274: L P[2274] 800cm/min CNT100 COORD PTH ;
:SR[23]=$SCR_GRP[1].$MCH_POS_X;
:SR[24]=$SCR_GRP[1].$MCH_POS_Y;
2275: L P[2275] 800cm/min CNT100 COORD PTH ;
:SR[23]=$SCR_GRP[1].$MCH_POS_X;
:SR[24]=$SCR_GRP[1].$MCH_POS_Y;
2276: L P[2276] 800cm/min CNT100 COORD PTH ;
:SR[23]=$SCR_GRP[1].$MCH_POS_X;
:SR[24]=$SCR_GRP[1].$MCH_POS_Y;
2277: L P[2277] 800cm/min CNT100 COORD PTH ;
:SR[23]=$SCR_GRP[1].$MCH_POS_X;
:SR[24]=$SCR_GRP[1].$MCH_POS_Y;
2278: L P[2278] 800cm/min CNT100 COORD PTH ;
:SR[23]=$SCR_GRP[1].$MCH_POS_X;
:SR[24]=$SCR_GRP[1].$MCH_POS_Y;
2279: L P[2279] 800cm/min CNT100 COORD PTH ;
:SR[23]=$SCR_GRP[1].$MCH_POS_X;
:SR[24]=$SCR_GRP[1].$MCH_POS_Y;
2280: L P[2280] 800cm/min CNT100 COORD PTH ;
:SR[23]=$SCR_GRP[1].$MCH_POS_X;
:SR[24]=$SCR_GRP[1].$MCH_POS_Y;
2281: L P[2281] 800cm/min CNT100 COORD PTH ;
:SR[23]=$SCR_GRP[1].$MCH_POS_X;
:SR[24]=$SCR_GRP[1].$MCH_POS_Y;
2282: L P[2282] 800cm/min CNT100 COORD PTH ;
:SR[23]=$SCR_GRP[1].$MCH_POS_X;
:SR[24]=$SCR_GRP[1].$MCH_POS_Y;
2283: L P[2283] 800cm/min CNT100 COORD PTH ;
:SR[23]=$SCR_GRP[1].$MCH_POS_X;
:SR[24]=$SCR_GRP[1].$MCH_POS_Y;
2284: L P[2284] 800cm/min CNT100 COORD PTH ;
:SR[23]=$SCR_GRP[1].$MCH_POS_X;
:SR[24]=$SCR_GRP[1].$MCH_POS_Y;
2285: L P[2285] 800cm/min CNT100 COORD PTH ;
:SR[23]=$SCR_GRP[1].$MCH_POS_X;
:SR[24]=$SCR_GRP[1].$MCH_POS_Y;
2286: L P[2286] 800cm/min CNT100 COORD PTH ;
:SR[23]=$SCR_GRP[1].$MCH_POS_X;
:SR[24]=$SCR_GRP[1].$MCH_POS_Y;
2287: L P[2287] 800cm/min CNT100 COORD PTH ;
:SR[23]=$SCR_GRP[1].$MCH_POS_X;
:SR[24]=$SCR_GRP[1].$MCH_POS_Y;
2288: L P[2288] 800cm/min CNT100 COORD PTH ;
:SR[23]=$SCR_GRP[1].$MCH_POS_X;
:SR[24]=$SCR_GRP[1].$MCH_POS_Y;
2289: L P[2289] 800cm/min CNT100 COORD PTH ;
:SR[23]=$SCR_GRP[1].$MCH_POS_X;
:SR[24]=$SCR_GRP[1].$MCH_POS_Y;
2290: L P[2290] 800cm/min CNT100 COORD PTH ;
:SR[23]=$SCR_GRP[1].$MCH_POS_X;
:SR[24]=$SCR_GRP[1].$MCH_POS_Y;
2291: L P[2291] 800cm/min CNT100 COORD PTH ;
:SR[23]=$SCR_GRP[1].$MCH_POS_X;
:SR[24]=$SCR_GRP[1].$MCH_POS_Y;
2292: L P[2292] 800cm/min CNT100 COORD PTH ;
:SR[23]=$SCR_GRP[1].$MCH_POS_X;
:SR[24]=$SCR_GRP[1].$MCH_POS_Y;
2293: L P[2293] 800cm/min CNT100 COORD PTH ;
:SR[23]=$SCR_GRP[1].$MCH_POS_X;
:SR[24]=$SCR_GRP[1].$MCH_POS_Y;
2294: L P[2294] 800cm/min CNT100 COORD PTH ;
:SR[23]=$SCR_GRP[1].$MCH_POS_X;
:SR[24]=$SCR_GRP[1].$MCH_POS_Y;
2295: L P[2295] 800cm/min CNT100 COORD PTH ;
:SR[23]=$SCR_GRP[1].$MCH_POS_X;
:SR[24]=$SCR_GRP[1].$MCH_POS_Y;
2296: L P[2296] 800cm/min CNT100 COORD PTH ;
:SR[23]=$SCR_GRP[1].$MCH_POS_X;
:SR[24]=$SCR_GRP[1].$MCH_POS_Y;
2297: L P[2297] 800cm/min CNT100 COORD PTH ;
:SR[23]=$SCR_GRP[1].$MCH_POS_X;
:SR[24]=$SCR_GRP[1].$MCH_POS_Y;
2298: L P[2298] 800cm/min CNT100 COORD PTH ;
:SR[23]=$SCR_GRP[1].$MCH_POS_X;
:SR[24]=$SCR_GRP[1].$MCH_POS_Y;
2299: L P[2299] 800cm/min CNT100 COORD PTH ;
:SR[23]=$SCR_GRP[1].$MCH_POS_X;
:SR[24]=$SCR_GRP[1].$MCH_POS_Y;
2300: L P[2300] 800cm/min CNT100 COORD PTH ;
:SR[23]=$SCR_GRP[1].$MCH_POS_X;
:SR[24]=$SCR_GRP[1].$MCH_POS_Y;
2301: L P[2301] 800cm/min CNT100 COORD PTH ;
:SR[23]=$SCR_GRP[1].$MCH_POS_X;
:SR[24]=$SCR_GRP[1].$MCH_POS_Y;
2302: L P[2302] 800cm/min CNT100 COORD PTH ;
:SR[23]=$SCR_GRP[1].$MCH_POS_X;
:SR[24]=$SCR_GRP[1].$MCH_POS_Y;
2303: L P[2303] 800cm/min CNT100 COORD PTH ;
:SR[23]=$SCR_GRP[1].$MCH_POS_X;
:SR[24]=$SCR_GRP[1].$MCH_POS_Y;
2304: L P[2304] 800cm/min CNT100 COORD PTH ;
:SR[23]=$SCR_GRP[1].$MCH_POS_X;
:SR[24]=$SCR_GRP[1].$MCH_POS_Y;
2305: L P[2305] 800cm/min CNT100 COORD PTH ;
:SR[23]=$SCR_GRP[1].$MCH_POS_X;
:SR[24]=$SCR_GRP[1].$MCH_POS_Y;
2306: L P[2306] 800cm/min CNT100 COORD PTH ;
:SR[23]=$SCR_GRP[1].$MCH_POS_X;
:SR[24]=$SCR_GRP[1].$MCH_POS_Y;
2307: L P[2307] 800cm/min CNT100 COORD PTH ;
:SR[23]=$SCR_GRP[1].$MCH_POS_X;
:SR[24]=$SCR_GRP[1].$MCH_POS_Y;
2308: L P[2308] 800cm/min CNT100 COORD PTH ;
:SR[23]=$SCR_GRP[1].$MCH_POS_X;
:SR[24]=$SCR_GRP[1].$MCH_POS_Y;
2309: L P[2309] 800cm/min CNT100 COORD PTH ;
:SR[23]=$SCR_GRP[1].$MCH_POS_X;
:SR[24]=$SCR_GRP[1].$MCH_POS_Y;
2310: L P[2310] 800cm/min CNT100 COORD PTH ;
:SR[23]=$SCR_GRP[1].$MCH_POS_X;
:SR[24]=$SCR_GRP[1].$MCH_POS_Y;
2311: L P[2311] 800cm/min CNT100 COORD PTH ;
:SR[23]=$SCR_GRP[1].$MCH_POS_X;
:SR[24]=$SCR_GRP[1].$MCH_POS_Y;
2312: L P[2312] 800cm/min CNT100 COORD PTH ;
:SR[23]=$SCR_GRP[1].$MCH_POS_X;
:SR[24]=$SCR_GRP[1].$MCH_POS_Y;
2313: L P[2313] 800cm/min CNT100 COORD PTH ;
:SR[23]=$SCR_GRP[1].$MCH_POS_X;
:SR[24]=$SCR_GRP[1].$MCH_POS_Y;
2314: L P[2314] 800cm/min CNT100 COORD PTH ;
:SR[23]=$SCR_GRP[1].$MCH_POS_X;
:SR[24]=$SCR_GRP[1].$MCH_POS_Y;
2315: L P[2315] 800cm/min CNT100 COORD PTH ;
:SR[23]=$SCR_GRP[1].$MCH_POS_X;
:SR[24]=$SCR_GRP[1].$MCH_POS_Y;
2316: L P[2316] 800cm/min CNT100 COORD PTH ;
:SR[23]=$SCR_GRP[1].$MCH_POS_X;
:SR[24]=$SCR_GRP[1].$MCH_POS_Y;
2317: L P[2317] 800cm/min CNT100 COORD PTH ;
:SR[23]=$SCR_GRP[1].$MCH_POS_X;
:SR[24]=$SCR_GRP[1].$MCH_POS_Y;
2318: L P[2318] 800cm/min CNT100 COORD PTH ;
:SR[23]=$SCR_GRP[1].$MCH_POS_X;
:SR[24]=$SCR_GRP[1].$MCH_POS_Y;
2319: L P[2319] 800cm/min CNT100 COORD PTH ;
:SR[23]=$SCR_GRP[1].$MCH_POS_X;
:SR[24]=$SCR_GRP[1].$MCH_POS_Y;
2320: L P[2320] 800cm/min CNT100 COORD PTH ;
:SR[23]=$SCR_GRP[1].$MCH_POS_X;
:SR[24]=$SCR_GRP[1].$MCH_POS_Y;
2321: L P[2321] 800cm/min CNT100 COORD PTH ;
:SR[23]=$SCR_GRP[1].$MCH_POS_X;
:SR[24]=$SCR_GRP[1].$MCH_POS_Y;
2322: L P[2322] 800cm/min CNT100 COORD PTH ;
:SR[23]=$SCR_GRP[1].$MCH_POS_X;
:SR[24]=$SCR_GRP[1].$MCH_POS_Y;
2323: L P[2323] 800cm/min CNT100 COORD PTH ;
:SR[23]=$SCR_GRP[1].$MCH_POS_X;
:SR[24]=$SCR_GRP[1].$MCH_POS_Y;
2324: L P[2324] 800cm/min CNT100 COORD PTH ;
:SR[23]=$SCR_GRP[1].$MCH_POS_X;
:SR[24]=$SCR_GRP[1].$MCH_POS_Y;
2325: L P[2325] 800cm/min CNT100 COORD PTH ;
:SR[23]=$SCR_GRP[1].$MCH_POS_X;
:SR[24]=$SCR_GRP[1].$MCH_POS_Y;
2326: L P[2326] 800cm/min CNT100 COORD PTH ;
:SR[23]=$SCR_GRP[1].$MCH_POS_X;
:SR[24]=$SCR_GRP[1].$MCH_POS_Y;
2327: L P[2327] 800cm/min CNT100 COORD PTH ;
:SR[23]=$SCR_GRP[1].$MCH_POS_X;
:SR[24]=$SCR_GRP[1].$MCH_POS_Y;
2328: L P[2328] 800cm/min CNT100 COORD PTH ;
:SR[23]=$SCR_GRP[1].$MCH_POS_X;
:SR[24]=$SCR_GRP[1].$MCH_POS_Y;
2329: L P[2329] 800cm/min CNT100 COORD PTH ;
:SR[23]=$SCR_GRP[1].$MCH_POS_X;
:SR[24]=$SCR_GRP[1].$MCH_POS_Y;
2330: L P[2330] 800cm/min CNT100 COORD PTH ;
:SR[23]=$SCR_GRP[1].$MCH_POS_X;
:SR[24]=$SCR_GRP[1].$MCH_POS_Y;
2331: L P[2331] 800cm/min CNT100 COORD PTH ;
:SR[23]=$SCR_GRP[1].$MCH_POS_X;
:SR[24]=$SCR_GRP[1].$MCH_POS_Y;
2332: L P[2332] 800cm/min CNT100 COORD PTH ;
:SR[23]=$SCR_GRP[1].$MCH_POS_X;
:SR[24]=$SCR_GRP[1].$MCH_POS_Y;
2333: L P[2333] 800cm/min CNT100 COORD PTH ;
:SR[23]=$SCR_GRP[1].$MCH_POS_X;
:SR[24]=$SCR_GRP[1].$MCH_POS_Y;
2334: L P[2334] 800cm/min CNT100 COORD PTH ;
:SR[23]=$SCR_GRP[1].$MCH_POS_X;
:SR[24]=$SCR_GRP[1].$MCH_POS_Y;
2335: L P[2335] 800cm/min CNT100 COORD PTH ;
:SR[23]=$SCR_GRP[1].$MCH_POS_X;
:SR[24]=$SCR_GRP[1].$MCH_POS_Y;
2336: L P[2336] 800cm/min CNT100 COORD PTH ;
:SR[23]=$SCR_GRP[1].$MCH_POS_X;
:SR[24]=$SCR_GRP[1].$MCH_POS_Y;
2337: L P[2337] 800cm/min CNT100 COORD PTH ;
:SR[23]=$SCR_GRP[1].$MCH_POS_X;
:SR[24]=$SCR_GRP[1].$MCH_POS_Y;
2338: L P[2338] 800cm/min CNT100 COORD PTH ;
:SR[23]=$SCR_GRP[1].$MCH_POS_X;
:SR[24]=$SCR_GRP[1].$MCH_POS_Y;
2339: L P[2339] 800cm/min CNT100 COORD PTH ;
:SR[23]=$SCR_GRP[1].$MCH_POS_X;
:SR[24]=$SCR_GRP[1].$MCH_POS_Y;
2340: L P[2340] 800cm/min CNT100 COORD PTH ;
:SR[23]=$SCR_GRP[1].$MCH_POS_X;
:SR[24]=$SCR_GRP[1].$MCH_POS_Y;
2341: L P[2341] 800cm/min CNT100 COORD PTH ;
:SR[23]=$SCR_GRP[1].$MCH_POS_X;
:SR[24]=$SCR_GRP[1].$MCH_POS_Y;
2342: L P[2342] 800cm/min CNT100 COORD PTH ;
:SR[23]=$SCR_GRP[1].$MCH_POS_X;
:SR[24]=$SCR_GRP[1].$MCH_POS_Y;
2343: L P[2343] 800cm/min CNT100 COORD PTH ;
:SR[23]=$SCR_GRP[1].$MCH_POS_X;
:SR[24]=$SCR_GRP[1].$MCH_POS_Y;
2344: L P[2344] 800cm/min CNT100 COORD PTH ;
:SR[23]=$SCR_GRP[1].$MCH_POS_X;
:SR[24]=$SCR_GRP[1].$MCH_POS_Y;
2345: L P[2345] 800cm/min CNT100 COORD PTH ;
:SR[23]=$SCR_GRP[1].$MCH_POS_X;
:SR[24]=$SCR_GRP[1].$MCH_POS_Y;
2346: L P[2346] 800cm/min CNT100 COORD PTH ;
:SR[23]=$SCR_GRP[1].$MCH_POS_X;
:SR[24]=$SCR_GRP[1].$MCH_POS_Y;
2347: L P[2347] 800cm/min CNT100 COORD PTH ;
:SR[23]=$SCR_GRP[1].$MCH_POS_X;
:SR[24]=$SCR_GRP[1].$MCH_POS_Y;
2348: L P[2348] 800cm/min CNT100 COORD PTH ;
:SR[23]=$SCR_GRP[1].$MCH_POS_X;
:SR[24]=$SCR_GRP[1].$MCH_POS_Y;
2349: L P[2349] 800cm/min CNT100 COORD PTH ;
:SR[23]=$SCR_GRP[1].$MCH_POS_X;
:SR[24]=$SCR_GRP[1].$MCH_POS_Y;
2350: L P[2350] 800cm/min CNT100 COORD PTH ;
:SR[23]=$SCR_GRP[1].$MCH_POS_X;
:SR[24]=$SCR_GRP[1].$MCH_POS_Y;
2351: L P[2351] 800cm/min CNT100 COORD PTH ;
:SR[23]=$SCR_GRP[1].$MCH_POS_X;
:SR[24]=$SCR_GRP[1].$MCH_POS_Y;
2352: L P[2352] 800cm/min CNT100 COORD PTH ;
:SR[23]=$SCR_GRP[1].$MCH_POS_X;
:SR[24]=$SCR_GRP[1].$MCH_POS_Y;
2353: L P[2353] 800cm/min CNT100 COORD PTH ;
:SR[23]=$SCR_GRP[1].$MCH_POS_X;
:SR[24]=$SCR_GRP[1].$MCH_POS_Y;
2354: L P[2354] 800cm/min CNT100 COORD PTH ;
:SR[23]=$SCR_GRP[1].$MCH_POS_X;
:SR[24]=$SCR_GRP[1].$MCH_POS_Y;
2355: L P[2355] 800cm/min CNT100 COORD PTH ;
:SR[23]=$SCR_GRP[1].$MCH_POS_X;
:SR[24]=$SCR_GRP[1].$MCH_POS_Y;
2356: L P[2356] 800cm/min CNT100 COORD PTH ;
:SR[23]=$SCR_GRP[1].$MCH_POS_X;
:SR[24]=$SCR_GRP[1].$MCH_POS_Y;
2357: L P[2357] 800cm/min CNT100 COORD PTH ;
:SR[23]=$SCR_GRP[1].$MCH_POS_X;
:SR[24]=$SCR_GRP[1].$MCH_POS_Y;
2358: L P[2358] 800cm/min CNT100 COORD PTH ;
:SR[23]=$SCR_GRP[1].$MCH_POS_X;
:SR[24]=$SCR_GRP[1].$MCH_POS_Y;
2359: L P[2359] 800cm/min CNT100 COORD PTH ;
:SR[23]=$SCR_GRP[1].$MCH_POS_X;
:SR[24]=$SCR_GRP[1].$MCH_POS_Y;
2360: L P[2360] 800cm/min CNT100 COORD PTH ;
:SR[23]=$SCR_GRP[1].$MCH_POS_X;
:SR[24]=$SCR_GRP[1].$MCH_POS_Y;
2361: L P[2361] 800cm/min CNT100 COORD PTH ;
:SR[23]=$SCR_GRP[1].$MCH_POS_X;
:SR[24]=$SCR_GRP[1].$MCH_POS_Y;
2362: L P[2362] 800cm/min CNT100 COORD PTH ;
:SR[23]=$SCR_GRP[1].$MCH_POS_X;
:SR[24]=$SCR_GRP[1].$MCH_POS_Y;
2363: L P[2363] 800cm/min CNT100 COORD PTH ;
:SR[23]=$SCR_GRP[1].$MCH_POS_X;
:SR[24]=$SCR_GRP[1].$MCH_POS_Y;
2364: L P[2364] 800cm/min CNT100 COORD PTH ;
:SR[23]=$SCR_GRP[1].$MCH_POS_X;
:SR[24]=$SCR_GRP[1].$MCH_POS_Y;
2365: L P[2365] 800cm/min CNT100 COORD PTH ;
:SR[23]=$SCR_GRP[1].$MCH_POS_X;
:SR[24]=$SCR_GRP[1].$MCH_POS_Y;
2366: L P[2366] 800cm/min CNT100 COORD PTH ;
:SR[23]=$SCR_GRP[1].$MCH_POS_X;
:SR[24]=$SCR_GRP[1].$MCH_POS_Y;
2367: L P[2367] 800cm/min CNT100 COORD PTH ;
:SR[23]=$SCR_GRP[1].$MCH_POS_X;
:SR[24]=$SCR_GRP[1].$MCH_POS_Y;
2368: L P[2368] 800cm/min CNT100 COORD PTH ;
:SR[23]=$SCR_GRP[1].$MCH_POS_X;
:SR[24]=$SCR_GRP[1].$MCH_POS_Y;
2369: L P[2369] 800cm/min CNT100 COORD PTH ;
:SR[23]=$SCR_GRP[1].$MCH_POS_X;
:SR[24]=$SCR_GRP[1].$MCH_POS_Y;
2370: L P[2370] 800cm/min CNT100 COORD PTH ;
:SR[23]=$SCR_GRP[1].$MCH_POS_X;
:SR[24]=$SCR_GRP[1].$MCH_POS_Y;
2371: L P[2371] 800cm/min CNT100 COORD PTH ;
:SR[23]=$SCR_GRP[1].$MCH_POS_X;
:SR[24]=$SCR_GRP[1].$MCH_POS_Y;
2372: L P[2372] 800cm/min CNT100 COORD PTH ;
:SR[23]=$SCR_GRP[1].$MCH_POS_X;
:SR[24]=$SCR_GRP[1].$MCH_POS_Y;
2373: L P[2373] 800cm/min CNT100 COORD PTH ;
:SR[23]=$SCR_GRP[1].$MCH_POS_X;
:SR[24]=$SCR_GRP[1].$MCH_POS_Y;
2374: L P[2374] 800cm/min CNT100 COORD PTH ;
:SR[23]=$SCR_GRP[1].$MCH_POS_X;
:SR[24]=$SCR_GRP[1].$MCH_POS_Y;
2375: L P[2375] 800cm/min CNT100 COORD PTH ;
:SR[23]=$SCR_GRP[1].$MCH_POS_X;
:SR[24]=$SCR_GRP[1].$MCH_POS_Y;
2376: L P[2376] 800cm/min CNT100 COORD PTH ;
:SR[23]=$SCR_GRP[1].$MCH_POS_X;
:SR[24]=$SCR_GRP[1].$MCH_POS_Y;
2377: L P[2377] 800cm/min CNT100 COORD PTH ;
:SR[23]=$SCR_GRP[1].$MCH_POS_X;
:SR[24]=$SCR_GRP[1].$MCH_POS_Y;
2378: L P[2378] 800cm/min CNT100 COORD PTH ;
:SR[23]=$SCR_GRP[1].$MCH_POS_X;
:SR[24]=$SCR_GRP[1].$MCH_POS_Y;
2379: L P[2379] 800cm/min CNT100 COORD PTH ;
:SR[23]=$SCR_GRP[1].$MCH_POS_X;
:SR[24]=$SCR_GRP[1].$MCH_POS_Y;
2380: L P[2380] 800cm/min CNT100 COORD PTH ;
:SR[23]=$SCR_GRP[1].$MCH_POS_X;
:SR[24]=$SCR_GRP[1].$MCH_POS_Y;
2381: L P[2381] 800cm/min CNT100 COORD PTH ;
:SR[23]=$SCR_GRP[1].$MCH_POS_X;
:SR[24]=$SCR_GRP[1].$MCH_POS_Y;
2382: L P[2382] 800cm/min CNT100 COORD PTH ;
:SR[23]=$SCR_GRP[1].$MCH_POS_X;
:SR[24]=$SCR_GRP[1].$MCH_POS_Y;
2383: L P[2383] 800cm/min CNT100 COORD PTH ;
:SR[23]=$SCR_GRP[1].$MCH_POS_X;
:SR[24]=$SCR_GRP[1].$MCH_POS_Y;
2384: L P[2384] 800cm/min CNT100 COORD PTH ;
:SR[23]=$SCR_GRP[1].$MCH_POS_X;
:SR[24]=$SCR_GRP[1].$MCH_POS_Y;
2385: L P[2385] 800cm/min CNT100 COORD PTH ;
:SR[23]=$SCR_GRP[1].$MCH_POS_X;
:SR[24]=$SCR_GRP[1].$MCH_POS_Y;
2386: L P[2386] 800cm/min CNT100 COORD PTH ;
:SR[23]=$SCR_GRP[1].$MCH_POS_X;
:SR[24]=$SCR_GRP[1].$MCH_POS_Y;
2387: L P[2387] 800cm/min CNT100 COORD PTH ;
:SR[23]=$SCR_GRP[1].$MCH_POS_X;
:SR[24]=$SCR_GRP[1].$MCH_POS_Y;
2388: L P[2388] 800cm/min CNT100 COORD PTH ;
:SR[23]=$SCR_GRP[1].$MCH_POS_X;
:SR[24]=$SCR_GRP[1].$MCH_POS_Y;
2389: L P[2389] 800cm/min CNT100 COORD PTH ;
:SR[23]=$SCR_GRP[1].$MCH_POS_X;
:SR[24]=$SCR_GRP[1].$MCH_POS_Y;
2390: L P[2390] 800cm/min CNT100 COORD PTH ;
:SR[23]=$SCR_GRP[1].$MCH_POS_X;
:SR[24]=$SCR_GRP[1].$MCH_POS_Y;
2391: L P[2391] 800cm/min CNT100 COORD PTH ;
:SR[23]=$SCR_GRP[1].$MCH_POS_X;
:SR[24]=$SCR_GRP[1].$MCH_POS_Y;
2392: L P[2392] 800cm/min CNT100 COORD PTH ;
:SR[23]=$SCR_GRP[1].$MCH_POS_X;
:SR[24]=$SCR_GRP[1].$MCH_POS_Y;
2393: L P[2393] 800cm/min CNT100 COORD PTH ;
:SR[23]=$SCR_GRP[1].$MCH_POS_X;
:SR[24]=$SCR_GRP[1].$MCH_POS_Y;
2394: L P[2394] 800cm/min CNT100 COORD PTH ;
:SR[23]=$SCR_GRP[1].$MCH_POS_X;
:SR[24]=$SCR_GRP[1].$MCH_POS_Y;
2395: L P[2395] 800cm/min CNT100 COORD PTH ;
:SR[23]=$SCR_GRP[1].$MCH_POS_X;
:SR[24]=$SCR_GRP[1].$MCH_POS_Y;
2396: L P[2396] 800cm/min CNT100 COORD PTH ;
:SR[23]=$SCR_GRP[1].$MCH_POS_X;
:SR[24]=$SCR_GRP[1].$MCH_POS_Y;
2397: L P[2397] 800cm/min CNT100 COORD PTH ;
:SR[23]=$SCR_GRP[1].$MCH_POS_X;
:SR[24]=$SCR_GRP[1].$MCH_POS_Y;
2398: L P[2398] 800cm/min CNT100 COORD PTH ;
:SR[23]=$SCR_GRP[1].$MCH_POS_X;
:SR[24]=$SCR_GRP[1].$MCH_POS_Y;
2399: L P[2399] 800cm/min CNT100 COORD PTH ;
:SR[23]=$SCR_GRP[1].$MCH_POS_X;
:SR[24]=$SCR_GRP[1].$MCH_POS_Y;
2400: L P[2400] 800cm/min CNT100 COORD PTH ;
:SR[23]=$SCR_GRP[1].$MCH_POS_X;
:SR[24]=$SCR_GRP[1].$MCH_POS_Y;
2401: L P[2401] 800cm/min CNT100 COORD PTH ;
:SR[23]=$SCR_GRP[1].$MCH_POS_X;
:SR[24]=$SCR_GRP[1].$MCH_POS_Y;
2402: L P[2402] 800cm/min CNT100 COORD PTH ;
:SR[23]=$SCR_GRP[1].$MCH_POS_X;
:SR[24]=$SCR_GRP[1].$MCH_POS_Y;
2403: L P[2403] 800cm/min CNT100 COORD PTH ;
:SR[23]=$SCR_GRP[1].$MCH_POS_X;
:SR[24]=$SCR_GRP[1].$MCH_POS_Y;
2404: L P[2404] 800cm/min CNT100 COORD PTH ;
:SR[23]=$SCR_GRP[1].$MCH_POS_X;
:SR[24]=$SCR_GRP[1].$MCH_POS_Y;
2405: L P[2405] 800cm/min CNT100 COORD PTH ;
:SR[23]=$SCR_GRP[1].$MCH_POS_X;
:SR[24]=$SCR_GRP[1].$MCH_POS_Y;
2406: L P[2406] 800cm/min CNT100 COORD PTH ;
:SR[23]=$SCR_GRP[1].$MCH_POS_X;
:SR[24]=$SCR_GRP[1].$MCH_POS_Y;
2407: L P[2407] 800cm/min CNT100 COORD PTH ;
:SR[23]=$SCR_GRP[1].$MCH_POS_X;
:SR[24]=$SCR_GRP[1].$MCH_POS_Y;
2408: L P[2408] 800cm/min CNT100 COORD PTH ;
:SR[23]=$SCR_GRP[1].$MCH_POS_X;
:SR[24]=$SCR_GRP[1].$MCH_POS_Y;
2409: L P[2409] 800cm/min CNT100 COORD PTH ;
:SR[23]=$SCR_GRP[1].$MCH_POS_X;
:SR[24]=$SCR_GRP[1].$MCH_POS_Y;
2410: L P[2410] 800cm/min CNT100 COORD PTH ;
:SR[23]=$SCR_GRP[1].$MCH_POS_X;
:SR[24]=$SCR_GRP[1].$MCH_POS_Y;
2411: L P[2411] 800cm/min CNT100 COORD PTH ;
:SR[23]=$SCR_GRP[1].$MCH_POS_X;
:SR[24]=$SCR_GRP[1].$MCH_POS_Y;
2412: L P[2412] 800cm/min CNT100 COORD PTH ;
:SR[23]=$SCR_GRP[1].$MCH_POS_X;
:SR[24]=$SCR_GRP[1].$MCH_POS_Y;
2413: L P[2413] 800cm/min CNT100 COORD PTH ;
:SR[23]=$SCR_GRP[1].$MCH_POS_X;
:SR[24]=$SCR_GRP[1].$MCH_POS_Y;
2414: L P[2414] 800cm/min CNT100 COORD PTH ;
:SR[23]=$SCR_GRP[1].$MCH_POS_X;
:SR[24]=$SCR_GRP[1].$MCH_POS_Y;
2415: L P[2415] 800cm/min CNT100 COORD PTH ;
:SR[23]=$SCR_GRP[1].$MCH_POS_X;
:SR[24]=$SCR_GRP[1].$MCH_POS_Y;
2416: L P[2416] 800cm/min CNT100 COORD PTH ;
:SR[23]=$SCR_GRP[1].$MCH_POS_X;
:SR[24]=$SCR_GRP[1].$MCH_POS_Y;
2417: L P[2417] 800cm/min CNT100 COORD PTH ;
:SR[23]=$SCR_GRP[1].$MCH_POS_X;
:SR[24]=$SCR_GRP[1].$MCH_POS_Y;
2418: L P[2418] 800cm/min CNT100 COORD PTH ;
:SR[23]=$SCR_GRP[1].$MCH_POS_X;
:SR[24]=$SCR_GRP[1].$MCH_POS_Y;
2419: L P[2419] 800cm/min CNT100 COORD PTH ;
:SR[23]=$SCR_GRP[1].$MCH_POS_X;
:SR[24]=$SCR_GRP[1].$MCH_POS_Y;
2420: L P[2420] 800cm/min CNT100 COORD PTH ;
:SR[23]=$SCR_GRP[1].$MCH_POS_X;
:SR[24]=$SCR_GRP[1].$MCH_POS_Y;
2421: L P[2421] 800cm/min CNT100 COORD PTH ;
:SR[23]=$SCR_GRP[1].$MCH_POS_X;
:SR[24]=$SCR_GRP[1].$MCH_POS_Y;
2422: L P[2422] 800cm/min CNT100 COORD PTH ;
:SR[23]=$SCR_GRP[1].$MCH_POS_X;
:SR[24]=$SCR_GRP[1].$MCH_POS_Y;
2423: L P[2423] 800cm/min CNT100 COORD PTH ;
:SR[23]=$SCR_GRP[1].$MCH_POS_X;
:SR[24]=$SCR_GRP[1].$MCH_POS_Y;
2424: L P[2424] 800cm/min CNT100 COORD PTH ;
:SR[23]=$SCR_GRP[1].$MCH_POS_X;
:SR[24]=$SCR_GRP[1].$MCH_POS_Y;
2425: L P[2425] 800cm/min CNT100 COORD PTH ;
:SR[23]=$SCR_GRP[1].$MCH_POS_X;
:SR[24]=$SCR_GRP[1].$MCH_POS_Y;
2426: L P[2426] 800cm/min CNT100 COORD PTH ;
:SR[23]=$SCR_GRP[1].$MCH_POS_X;
:SR[24]=$SCR_GRP[1].$MCH_POS_Y;
2427: L P[2427] 800cm/min CNT100 COORD PTH ;
:SR[23]=$SCR_GRP[1].$MCH_POS_X;
:SR[24]=$SCR_GRP[1].$MCH_POS_Y;
2428: L P[2428] 800cm/min CNT100 COORD PTH ;
:SR[23]=$SCR_GRP[1].$MCH_POS_X;
:SR[24]=$SCR_GRP[1].$MCH_POS_Y;
2429: L P[2429] 800cm/min CNT100 COORD PTH ;
:SR[23]=$SCR_GRP[1].$MCH_POS_X;
:SR[24]=$SCR_GRP[1].$MCH_POS_Y;
2430: L P[2430] 800cm/min CNT100 COORD PTH ;
:SR[23]=$SCR_GRP[1].$MCH_POS_X;
:SR[24]=$SCR_GRP[1].$MCH_POS_Y;
2431: L P[2431] 800cm/min CNT100 COORD PTH ;
:SR[23]=$SCR_GRP[1].$MCH_POS_X;
:SR[24]=$SCR_GRP[1].$MCH_POS_Y;
2432: L P[2432] 800cm/min CNT100 COORD PTH ;
:SR[23]=$SCR_GRP[1].$MCH_POS_X;
:SR[24]=$SCR_GRP[1].$MCH_POS_Y;
2433: L P[2433] 800cm/min CNT100 COORD PTH ;
:SR[23]=$SCR_GRP[1].$MCH_POS_X;
:SR[24]=$SCR_GRP[1].$MCH_POS_Y;
2434: L P[2434] 800cm/min CNT100 COORD PTH ;
:SR[23]=$SCR_GRP[1].$MCH_POS_X;
:SR[24]=$SCR_GRP[1].$MCH_POS_Y;
2435: L P[2435] 800cm/min CNT100 COORD PTH ;
:SR[23]=$SCR_GRP[1].$MCH_POS_X;
:SR[24]=$SCR_GRP[1].$MCH_POS_Y;
2436: L P[2436] 800cm/min CNT100 COORD PTH ;
:SR[23]=$SCR_GRP[1].$MCH_POS_X;
:SR[24]=$SCR_GRP[1].$MCH_POS_Y;
2437: L P[2437] 800cm/min CNT100 COORD PTH ;
:SR[23]=$SCR_GRP[1].$MCH_POS_X;
:SR[24]=$SCR_GRP[1].$MCH_POS_Y;
2438: L P[2438] 800cm/min CNT100 COORD PTH ;
:SR[23]=$SCR_GRP[1].$MCH_POS_X;
:SR[24]=$SCR_GRP[1].$MCH_POS_Y;
2439: L P[2439] 800cm/min CNT100 COORD PTH ;
:SR[23]=$SCR_GRP[1].$MCH_POS_X;
:SR[24]=$SCR_GRP[1].$MCH_POS_Y;
2440: L P[2440] 800cm/min CNT100 COORD PTH ;
:SR[23]=$SCR_GRP[1].$MCH_POS_X;
:SR[24]=$SCR_GRP[1].$MCH_POS_Y;
2441: L P[2441] 800cm/min CNT100 COORD PTH ;
:SR[23]=$SCR_GRP[1].$MCH_POS_X;
:SR[24]=$SCR_GRP[1].$MCH_POS_Y;
2442: L P[2442] 800cm/min CNT100 COORD PTH ;
:SR[23]=$SCR_GRP[1].$MCH_POS_X;
:SR[24]=$SCR_GRP[1].$MCH_POS_Y;
2443: L P[2443] 800cm/min CNT100 COORD PTH ;
:SR[23]=$SCR_GRP[1].$MCH_POS_X;
:SR[24]=$SCR_GRP[1].$MCH_POS_Y;
2444: L P[2444] 800cm/min CNT100 COORD PTH ;
:SR[23]=$SCR_GRP[1].$MCH_POS_X;
:SR[24]=$SCR_GRP[1].$MCH_POS_Y;
2445: L P[2445] 800cm/min CNT100 COORD PTH ;
:SR[23]=$SCR_GRP[1].$MCH_POS_X;
:SR[24]=$SCR_GRP[1].$MCH_POS_Y;
2446: L P[2446] 800cm/min CNT100 COORD PTH ;
:SR[23]=$SCR_GRP[1].$MCH_POS_X;
:SR[24]=$SCR_GRP[1].$MCH_POS_Y;
2447: L P[2447] 800cm/min CNT100 COORD PTH ;
:SR[23]=$SCR_GRP[1].$MCH_POS_X;
:SR[24]=$SCR_GRP[1].$MCH_POS_Y;
2448: L P[2448] 800cm/min CNT100 COORD PTH ;
:SR[23]=$SCR_GRP[1].$MCH_POS_X;
:SR[24]=$SCR_GRP[1].$MCH_POS_Y;
2449: L P[2449] 800cm/min CNT100 COORD PTH ;
:SR[23]=$SCR_GRP[1].$MCH_POS_X;
:SR[24]=$SCR_GRP[1].$MCH_POS_Y;
2450: L P[2450] 800cm/min CNT100 COORD PTH ;
:SR[23]=$SCR_GRP[1].$MCH_POS_X;
:SR[24]=$SCR_GRP[1].$MCH_POS_Y;
2451: L P[2451] 800cm/min CNT100 COORD PTH ;
:SR[23]=$SCR_GRP[1].$MCH_POS_X;
:SR[24]=$SCR_GRP[1].$MCH_POS_Y;
2452: L P[2452] 800cm/min CNT100 COORD PTH ;
:SR[23]=$SCR_GRP[1].$MCH_POS_X;
:SR[24]=$SCR_GRP[1].$MCH_POS_Y;
2453: L P[2453] 800cm/min CNT100 COORD PTH ;
:SR[23]=$SCR_GRP[1].$MCH_POS_X;
:SR[24]=$SCR_GRP[1].$MCH_POS_Y;
2454: L P[2454] 800cm/min CNT100 COORD PTH ;
:SR[23]=$SCR_GRP[1].$MCH_POS_X;
:SR[24]=$SCR_GRP[1].$MCH_POS_Y;
2455: L P[2455] 800cm/min CNT100 COORD PTH ;
:SR[23]=$SCR_GRP[1].$MCH_POS_X;
:SR[24]=$SCR_GRP[1].$MCH_POS_Y;
2456: L P[2456] 800cm/min CNT100 COORD PTH ;
:SR[23]=$SCR_GRP[1].$MCH_POS_X;
:SR[24]=$SCR_GRP[1].$MCH_POS_Y;
2457: L P[2457] 800cm/min CNT100 COORD PTH ;
:SR[23]=$SCR_GRP[1].$MCH_POS_X;
:SR[24]=$SCR_GRP[1].$MCH_POS_Y;
2458: L P[2458] 800cm/min CNT100 COORD PTH ;
:SR[23]=$SCR_GRP[1].$MCH_POS_X;
:SR[24]=$SCR_GRP[1].$MCH_POS_Y;
2459: L P[2459] 800cm/min CNT100 COORD PTH ;
:SR[23]=$SCR_GRP[1].$MCH_POS_X;
:SR[24]=$SCR_GRP[1].$MCH_POS_Y;
2460: L P[2460] 800cm/min CNT100 COORD PTH ;
:SR[23]=$SCR_GRP[1].$MCH_POS_X;
:SR[24]=$SCR_GRP[1].$MCH_POS_Y;
2461: L P[2461] 800cm/min CNT100 COORD PTH ;
:SR[23]=$SCR_GRP[1].$MCH_POS_X;
:SR[24]=$SCR_GRP[1].$MCH_POS_Y;
2462: L P[2462] 800cm/min CNT100 COORD PTH ;
:SR[23]=$SCR_GRP[1].$MCH_POS_X;
:SR[24]=$SCR_GRP[1].$MCH_POS_Y;
2463: L P[2463] 800cm/min CNT100 COORD PTH ;
:SR[23]=$SCR_GRP[1].$MCH_POS_X;
:SR[24]=$SCR_GRP[1].$MCH_POS_Y;
2464: L P[2464] 800cm/min CNT100 COORD PTH ;
:SR[23]=$SCR_GRP[1].$MCH_POS_X;
:SR[24]=$SCR_GRP[1].$MCH_POS_Y;
2465: L P[2465] 800cm/min CNT100 COORD PTH ;
:SR[23]=$SCR_GRP[1].$MCH_POS_X;
:SR[24]=$SCR_GRP[1].$MCH_POS_Y;
2466: L P[2466] 800cm/min CNT100 COORD PTH ;
:SR[23]=$SCR_GRP[1].$MCH_POS_X;
:SR[24]=$SCR_GRP[1].$MCH_POS_Y;
2467: L P[2467] 800cm/min CNT100 COORD PTH ;
:SR[23]=$SCR_GRP[1].$MCH_POS_X;
:SR[24]=$SCR_GRP[1].$MCH_POS_Y;
2468: L P[2468] 800cm/min CNT100 COORD PTH ;
:SR[23]=$SCR_GRP[1].$MCH_POS_X;
:SR[24]=$SCR_GRP[1].$MCH_POS_Y;
2469: L P[2469] 800cm/min CNT100 COORD PTH ;
:SR[23]=$SCR_GRP[1].$MCH_POS_X;
:SR[24]=$SCR_GRP[1].$MCH_POS_Y;
2470: L P[2470] 800cm/min CNT100 COORD PTH ;
:SR[23]=$SCR_GRP[1].$MCH_POS_X;
:SR[24]=$SCR_GRP[1].$MCH_POS_Y;
2471: L P[2471] 800cm/min CNT100 COORD PTH ;
:SR[23]=$SCR_GRP[1].$MCH_POS_X;
:SR[24]=$SCR_GRP[1].$MCH_POS_Y;
2472: L P[2472] 800cm/min CNT100 COORD PTH ;
:SR[23]=$SCR_GRP[1].$MCH_POS_X;
:SR[24]=$SCR_GRP[1].$MCH_POS_Y;
2473: L P[2473] 800cm/min CNT100 COORD PTH ;
:SR[23]=$SCR_GRP[1].$MCH_POS_X;
:SR[24]=$SCR_GRP[1].$MCH_POS_Y;
2474: L P[2474] 800cm/min CNT100 COORD PTH ;
:SR[23]=$SCR_GRP[1].$MCH_POS_X;
:SR[24]=$SCR_GRP[1].$MCH_POS_Y;
2475: L P[2475] 800cm/min CNT100 COORD PTH ;
:SR[23]=$SCR_GRP[1].$MCH_POS_X;
:SR[24]=$SCR_GRP[1].$MCH_POS_Y;
2476: L P[2476] 800cm/min CNT100 COORD PTH ;
:SR[23]=$SCR_GRP[1].$MCH_POS_X;
:SR[24]=$SCR_GRP[1].$MCH_POS_Y;
2477: L P[2477] 800cm/min CNT100 COORD PTH ;
:SR[23]=$SCR_GRP[1].$MCH_POS_X;
:SR[24]=$SCR_GRP[1].$MCH_POS_Y;
2478: L P[2478] 800cm/min CNT100 COORD PTH ;
:SR[23]=$SCR_GRP[1].$MCH_POS_X;
:SR[24]=$SCR_GRP[1].$MCH_POS_Y;
2479: L P[2479] 800cm/min CNT100 COORD PTH ;
:SR[23]=$SCR_GRP[1].$MCH_POS_X;
:SR[24]=$SCR_GRP[1].$MCH_POS_Y;
2480: L P[2480] 800cm/min CNT100 COORD PTH ;
:SR[23]=$SCR_GRP[1].$MCH_POS_X;
:SR[24]=$SCR_GRP[1].$MCH_POS_Y;
2481: L P[2481] 800cm/min CNT100 COORD PTH ;
:SR[23]=$SCR_GRP[1].$MCH_POS_X;
:SR[24]=$SCR_GRP[1].$MCH_POS_Y;
2482: L P[2482] 800cm/min CNT100 COORD PTH ;
:SR[23]=$SCR_GRP[1].$MCH_POS_X;
:SR[24]=$SCR_GRP[1].$MCH_POS_Y;
2483: L P[2483] 800cm/min CNT100 COORD PTH ;
:SR[23]=$SCR_GRP[1].$MCH_POS_X;
:SR[24]=$SCR_GRP[1].$MCH_POS_Y;
2484: L P[2484] 800cm/min CNT100 COORD PTH ;
:SR[23]=$SCR_GRP[1].$MCH_POS_X;
:SR[24]=$SCR_GRP[1].$MCH_POS_Y;
2485: L P[2485] 800cm/min CNT100 COORD PTH ;
:SR[23]=$SCR_GRP[1].$MCH_POS_X;
:SR[24]=$SCR_GRP[1].$MCH_POS_Y;
2486: L P[2486] 800cm/min CNT100 COORD PTH ;
:SR[23]=$SCR_GRP[1].$MCH_POS_X;
:SR[24]=$SCR_GRP[1].$MCH_POS_Y;
2487: L P[2487] 800cm/min CNT100 COORD PTH ;
:SR[23]=$SCR_GRP[1].$MCH_POS_X;
:SR[24]=$SCR_GRP[1].$MCH_POS_Y;
2488: L P[2488] 800cm/min CNT100 COORD PTH ;
:SR[23]=$SCR_GRP[1].$MCH_POS_X;
:SR[24]=$SCR_GRP[1].$MCH_POS_Y;
2489: L P[2489] 800cm/min CNT100 COORD PTH ;
:SR[23]=$SCR_GRP[1].$MCH_POS_X;
:SR[24]=$SCR_GRP[1].$MCH_POS_Y;
2490: L P[2490] 800cm/min CNT100 COORD PTH ;
:SR[23]=$SCR_GRP[1].$MCH_POS_X;
:SR[24]=$SCR_GRP[1].$MCH_POS_Y;
2491: L P[2491] 800cm/min CNT100 COORD PTH ;
:SR[23]=$SCR_GRP[1].$MCH_POS_X;
:SR[24]=$SCR_GRP[1].$MCH_POS_Y;
2492: L P[2492] 800cm/min CNT100 COORD PTH ;
:SR[23]=$SCR_GRP[1].$MCH_POS_X;
:SR[24]=$SCR_GRP[1].$MCH_POS_Y;
2493: L P[2493] 800cm/min CNT100 COORD PTH ;
:SR[23]=$SCR_GRP[1].$MCH_POS_X;
:SR[24]=$SCR_GRP[1].$MCH_POS_Y;
2494: L P[2494] 800cm/min CNT100 COORD PTH ;
:SR[23]=$SCR_GRP[1].$MCH_POS_X;
:SR[24]=$SCR_GRP[1].$MCH_POS_Y;
2495: L P[2495] 800cm/min CNT100 COORD PTH ;
:SR[23]=$SCR_GRP[1].$MCH_POS_X;
:SR[24]=$SCR_GRP[1].$MCH_POS_Y;
2496: L P[2496] 800cm/min CNT100 COORD PTH ;
:SR[23]=$SCR_GRP[1].$MCH_POS_X;
:SR[24]=$SCR_GRP[1].$MCH_POS_Y;
2497: L P[2497] 800cm/min CNT100 COORD PTH ;
:SR[23]=$SCR_GRP[1].$MCH_POS_X;
:SR[24]=$SCR_GRP[1].$MCH_POS_Y;
2498: L P[2498] 800cm/min CNT100 COORD PTH ;
:SR[23]=$SCR_GRP[1].$MCH_POS_X;
:SR[24]=$SCR_GRP[1].$MCH_POS_Y;
2499: L P[2499] 800cm/min CNT100 COORD ;
:SR[23]=$SCR_GRP[1].$MCH_POS_X;
:SR[24]=$SCR_GRP[1].$MCH_POS_Y;
2500: L P[2500] 800cm/min CNT100 COORD PTH ;
:SR[23]=$SCR_GRP[1].$MCH_POS_X;
:SR[24]=$SCR_GRP[1].$MCH_POS_Y;
2501: L P[2501] 800cm/min CNT100 COORD PTH ;
:SR[23]=$SCR_GRP[1].$MCH_POS_X;
:SR[24]=$SCR_GRP[1].$MCH_POS_Y;
2502: L P[2502] 800cm/min CNT100 COORD PTH ;
:SR[23]=$SCR_GRP[1].$MCH_POS_X;
:SR[24]=$SCR_GRP[1].$MCH_POS_Y;
2503: L P[2503] 800cm/min CNT100 COORD PTH ;
:SR[23]=$SCR_GRP[1].$MCH_POS_X;
:SR[24]=$SCR_GRP[1].$MCH_POS_Y;
2504: L P[2504] 800cm/min CNT100 COORD PTH ;
:SR[23]=$SCR_GRP[1].$MCH_POS_X;
:SR[24]=$SCR_GRP[1].$MCH_POS_Y;
2505: L P[2505] 800cm/min CNT100 COORD PTH ;
:SR[23]=$SCR_GRP[1].$MCH_POS_X;
:SR[24]=$SCR_GRP[1].$MCH_POS_Y;
2506: L P[2506] 800cm/min CNT100 COORD PTH ;
:SR[23]=$SCR_GRP[1].$MCH_POS_X;
:SR[24]=$SCR_GRP[1].$MCH_POS_Y;
2507: L P[2507] 800cm/min CNT100 COORD PTH ;
:SR[23]=$SCR_GRP[1].$MCH_POS_X;
:SR[24]=$SCR_GRP[1].$MCH_POS_Y;
2508: L P[2508] 800cm/min CNT100 COORD PTH ;
:SR[23]=$SCR_GRP[1].$MCH_POS_X;
:SR[24]=$SCR_GRP[1].$MCH_POS_Y;
2509: L P[2509] 800cm/min CNT100 COORD PTH ;
:SR[23]=$SCR_GRP[1].$MCH_POS_X;
:SR[24]=$SCR_GRP[1].$MCH_POS_Y;
2510: L P[2510] 800cm/min CNT100 COORD PTH ;
:SR[23]=$SCR_GRP[1].$MCH_POS_X;
:SR[24]=$SCR_GRP[1].$MCH_POS_Y;
2511: L P[2511] 800cm/min CNT100 COORD PTH ;
:SR[23]=$SCR_GRP[1].$MCH_POS_X;
:SR[24]=$SCR_GRP[1].$MCH_POS_Y;
2512: L P[2512] 800cm/min CNT100 COORD PTH ;
:SR[23]=$SCR_GRP[1].$MCH_POS_X;
:SR[24]=$SCR_GRP[1].$MCH_POS_Y;
2513: L P[2513] 800cm/min CNT100 COORD PTH ;
:SR[23]=$SCR_GRP[1].$MCH_POS_X;
:SR[24]=$SCR_GRP[1].$MCH_POS_Y;
2514: L P[2514] 800cm/min CNT100 COORD PTH ;
:SR[23]=$SCR_GRP[1].$MCH_POS_X;
:SR[24]=$SCR_GRP[1].$MCH_POS_Y;
2515: L P[2515] 800cm/min CNT100 COORD PTH ;
:SR[23]=$SCR_GRP[1].$MCH_POS_X;
:SR[24]=$SCR_GRP[1].$MCH_POS_Y;
2516: L P[2516] 800cm/min CNT100 COORD PTH ;
:SR[23]=$SCR_GRP[1].$MCH_POS_X;
:SR[24]=$SCR_GRP[1].$MCH_POS_Y;
2517: L P[2517] 800cm/min CNT100 COORD PTH ;
:SR[23]=$SCR_GRP[1].$MCH_POS_X;
:SR[24]=$SCR_GRP[1].$MCH_POS_Y;
2518: L P[2518] 800cm/min CNT100 COORD PTH ;
:SR[23]=$SCR_GRP[1].$MCH_POS_X;
:SR[24]=$SCR_GRP[1].$MCH_POS_Y;
2519: L P[2519] 800cm/min CNT100 COORD PTH ;
:SR[23]=$SCR_GRP[1].$MCH_POS_X;
:SR[24]=$SCR_GRP[1].$MCH_POS_Y;
2520: L P[2520] 800cm/min CNT100 COORD PTH ;
:SR[23]=$SCR_GRP[1].$MCH_POS_X;
:SR[24]=$SCR_GRP[1].$MCH_POS_Y;
2521: L P[2521] 800cm/min CNT100 COORD PTH ;
:SR[23]=$SCR_GRP[1].$MCH_POS_X;
:SR[24]=$SCR_GRP[1].$MCH_POS_Y;
2522: L P[2522] 800cm/min CNT100 COORD PTH ;
:SR[23]=$SCR_GRP[1].$MCH_POS_X;
:SR[24]=$SCR_GRP[1].$MCH_POS_Y;
2523: L P[2523] 800cm/min CNT100 COORD PTH ;
:SR[23]=$SCR_GRP[1].$MCH_POS_X;
:SR[24]=$SCR_GRP[1].$MCH_POS_Y;
2524: L P[2524] 800cm/min CNT100 COORD PTH ;
:SR[23]=$SCR_GRP[1].$MCH_POS_X;
:SR[24]=$SCR_GRP[1].$MCH_POS_Y;
2525: L P[2525] 800cm/min CNT100 COORD PTH ;
:SR[23]=$SCR_GRP[1].$MCH_POS_X;
:SR[24]=$SCR_GRP[1].$MCH_POS_Y;
2526: L P[2526] 800cm/min CNT100 COORD PTH ;
:SR[23]=$SCR_GRP[1].$MCH_POS_X;
:SR[24]=$SCR_GRP[1].$MCH_POS_Y;
2527: L P[2527] 800cm/min CNT100 COORD PTH ;
:SR[23]=$SCR_GRP[1].$MCH_POS_X;
:SR[24]=$SCR_GRP[1].$MCH_POS_Y;
2528: L P[2528] 800cm/min CNT100 COORD PTH ;
:SR[23]=$SCR_GRP[1].$MCH_POS_X;
:SR[24]=$SCR_GRP[1].$MCH_POS_Y;
2529: L P[2529] 800cm/min CNT100 COORD PTH ;
:SR[23]=$SCR_GRP[1].$MCH_POS_X;
:SR[24]=$SCR_GRP[1].$MCH_POS_Y;
2530: L P[2530] 800cm/min CNT100 COORD PTH ;
:SR[23]=$SCR_GRP[1].$MCH_POS_X;
:SR[24]=$SCR_GRP[1].$MCH_POS_Y;
2531: L P[2531] 800cm/min CNT100 COORD PTH ;
:SR[23]=$SCR_GRP[1].$MCH_POS_X;
:SR[24]=$SCR_GRP[1].$MCH_POS_Y;
2532: L P[2532] 800cm/min CNT100 COORD PTH ;
:SR[23]=$SCR_GRP[1].$MCH_POS_X;
:SR[24]=$SCR_GRP[1].$MCH_POS_Y;
2533: L P[2533] 800cm/min CNT100 COORD PTH ;
:SR[23]=$SCR_GRP[1].$MCH_POS_X;
:SR[24]=$SCR_GRP[1].$MCH_POS_Y;
2534: L P[2534] 800cm/min CNT100 COORD PTH ;
:SR[23]=$SCR_GRP[1].$MCH_POS_X;
:SR[24]=$SCR_GRP[1].$MCH_POS_Y;
2535: L P[2535] 800cm/min CNT100 COORD PTH ;
:SR[23]=$SCR_GRP[1].$MCH_POS_X;
:SR[24]=$SCR_GRP[1].$MCH_POS_Y;
2536: L P[2536] 800cm/min CNT100 COORD PTH ;
:SR[23]=$SCR_GRP[1].$MCH_POS_X;
:SR[24]=$SCR_GRP[1].$MCH_POS_Y;
2537: L P[2537] 800cm/min CNT100 COORD PTH ;
:SR[23]=$SCR_GRP[1].$MCH_POS_X;
:SR[24]=$SCR_GRP[1].$MCH_POS_Y;
2538: L P[2538] 800cm/min CNT100 COORD PTH ;
:SR[23]=$SCR_GRP[1].$MCH_POS_X;
:SR[24]=$SCR_GRP[1].$MCH_POS_Y;
2539: L P[2539] 800cm/min CNT100 COORD PTH ;
:SR[23]=$SCR_GRP[1].$MCH_POS_X;
:SR[24]=$SCR_GRP[1].$MCH_POS_Y;
2540: L P[2540] 800cm/min CNT100 COORD PTH ;
:SR[23]=$SCR_GRP[1].$MCH_POS_X;
:SR[24]=$SCR_GRP[1].$MCH_POS_Y;
2541: L P[2541] 800cm/min CNT100 COORD PTH ;
:SR[23]=$SCR_GRP[1].$MCH_POS_X;
:SR[24]=$SCR_GRP[1].$MCH_POS_Y;
2542: L P[2542] 800cm/min CNT100 COORD PTH ;
:SR[23]=$SCR_GRP[1].$MCH_POS_X;
:SR[24]=$SCR_GRP[1].$MCH_POS_Y;
2543: L P[2543] 800cm/min CNT100 COORD PTH ;
:SR[23]=$SCR_GRP[1].$MCH_POS_X;
:SR[24]=$SCR_GRP[1].$MCH_POS_Y;
2544: L P[2544] 800cm/min CNT100 COORD PTH ;
:SR[23]=$SCR_GRP[1].$MCH_POS_X;
:SR[24]=$SCR_GRP[1].$MCH_POS_Y;
2545: L P[2545] 800cm/min CNT100 COORD PTH ;
:SR[23]=$SCR_GRP[1].$MCH_POS_X;
:SR[24]=$SCR_GRP[1].$MCH_POS_Y;
2546: L P[2546] 800cm/min CNT100 COORD PTH ;
:SR[23]=$SCR_GRP[1].$MCH_POS_X;
:SR[24]=$SCR_GRP[1].$MCH_POS_Y;
2547: L P[2547] 800cm/min CNT100 COORD PTH ;
:SR[23]=$SCR_GRP[1].$MCH_POS_X;
:SR[24]=$SCR_GRP[1].$MCH_POS_Y;
2548: L P[2548] 800cm/min CNT100 COORD PTH ;
:SR[23]=$SCR_GRP[1].$MCH_POS_X;
:SR[24]=$SCR_GRP[1].$MCH_POS_Y;
2549: L P[2549] 800cm/min CNT100 COORD PTH ;
:SR[23]=$SCR_GRP[1].$MCH_POS_X;
:SR[24]=$SCR_GRP[1].$MCH_POS_Y;
2550: L P[2550] 800cm/min CNT100 COORD PTH ;
:SR[23]=$SCR_GRP[1].$MCH_POS_X;
:SR[24]=$SCR_GRP[1].$MCH_POS_Y;
2551: L P[2551] 800cm/min CNT100 COORD PTH ;
:SR[23]=$SCR_GRP[1].$MCH_POS_X;
:SR[24]=$SCR_GRP[1].$MCH_POS_Y;
2552: L P[2552] 800cm/min CNT100 COORD PTH ;
:SR[23]=$SCR_GRP[1].$MCH_POS_X;
:SR[24]=$SCR_GRP[1].$MCH_POS_Y;
2553: L P[2553] 800cm/min CNT100 COORD PTH ;
:SR[23]=$SCR_GRP[1].$MCH_POS_X;
:SR[24]=$SCR_GRP[1].$MCH_POS_Y;
2554: L P[2554] 800cm/min CNT100 COORD PTH ;
:SR[23]=$SCR_GRP[1].$MCH_POS_X;
:SR[24]=$SCR_GRP[1].$MCH_POS_Y;
2555: L P[2555] 800cm/min CNT100 COORD PTH ;
:SR[23]=$SCR_GRP[1].$MCH_POS_X;
:SR[24]=$SCR_GRP[1].$MCH_POS_Y;
2556: L P[2556] 800cm/min CNT100 COORD PTH ;
:SR[23]=$SCR_GRP[1].$MCH_POS_X;
:SR[24]=$SCR_GRP[1].$MCH_POS_Y;
2557: L P[2557] 800cm/min CNT100 COORD PTH ;
:SR[23]=$SCR_GRP[1].$MCH_POS_X;
:SR[24]=$SCR_GRP[1].$MCH_POS_Y;
2558: L P[2558] 800cm/min CNT100 COORD PTH ;
:SR[23]=$SCR_GRP[1].$MCH_POS_X;
:SR[24]=$SCR_GRP[1].$MCH_POS_Y;
2559: L P[2559] 800cm/min CNT100 COORD PTH ;
:SR[23]=$SCR_GRP[1].$MCH_POS_X;
:SR[24]=$SCR_GRP[1].$MCH_POS_Y;
2560: L P[2560] 800cm/min CNT100 COORD PTH ;
:SR[23]=$SCR_GRP[1].$MCH_POS_X;
:SR[24]=$SCR_GRP[1].$MCH_POS_Y;
2561: L P[2561] 800cm/min CNT100 COORD PTH ;
:SR[23]=$SCR_GRP[1].$MCH_POS_X;
:SR[24]=$SCR_GRP[1].$MCH_POS_Y;
2562: L P[2562] 800cm/min CNT100 COORD PTH ;
:SR[23]=$SCR_GRP[1].$MCH_POS_X;
:SR[24]=$SCR_GRP[1].$MCH_POS_Y;
2563: L P[2563] 800cm/min CNT100 COORD PTH ;
:SR[23]=$SCR_GRP[1].$MCH_POS_X;
:SR[24]=$SCR_GRP[1].$MCH_POS_Y;
2564: L P[2564] 800cm/min CNT100 COORD PTH ;
:SR[23]=$SCR_GRP[1].$MCH_POS_X;
:SR[24]=$SCR_GRP[1].$MCH_POS_Y;
2565: L P[2565] 800cm/min CNT100 COORD PTH ;
:SR[23]=$SCR_GRP[1].$MCH_POS_X;
:SR[24]=$SCR_GRP[1].$MCH_POS_Y;
2566: L P[2566] 800cm/min CNT100 COORD PTH ;
:SR[23]=$SCR_GRP[1].$MCH_POS_X;
:SR[24]=$SCR_GRP[1].$MCH_POS_Y;
2567: L P[2567] 800cm/min CNT100 COORD PTH ;
:SR[23]=$SCR_GRP[1].$MCH_POS_X;
:SR[24]=$SCR_GRP[1].$MCH_POS_Y;
2568: L P[2568] 800cm/min CNT100 COORD PTH ;
:SR[23]=$SCR_GRP[1].$MCH_POS_X;
:SR[24]=$SCR_GRP[1].$MCH_POS_Y;
2569: L P[2569] 800cm/min CNT100 COORD PTH ;
:SR[23]=$SCR_GRP[1].$MCH_POS_X;
:SR[24]=$SCR_GRP[1].$MCH_POS_Y;
2570: L P[2570] 800cm/min CNT100 COORD PTH ;
:SR[23]=$SCR_GRP[1].$MCH_POS_X;
:SR[24]=$SCR_GRP[1].$MCH_POS_Y;
2571: L P[2571] 800cm/min CNT100 COORD PTH ;
:SR[23]=$SCR_GRP[1].$MCH_POS_X;
:SR[24]=$SCR_GRP[1].$MCH_POS_Y;
2572: L P[2572] 800cm/min CNT100 COORD PTH ;
:SR[23]=$SCR_GRP[1].$MCH_POS_X;
:SR[24]=$SCR_GRP[1].$MCH_POS_Y;
2573: L P[2573] 800cm/min CNT100 COORD PTH ;
:SR[23]=$SCR_GRP[1].$MCH_POS_X;
:SR[24]=$SCR_GRP[1].$MCH_POS_Y;
2574: L P[2574] 800cm/min CNT100 COORD PTH ;
:SR[23]=$SCR_GRP[1].$MCH_POS_X;
:SR[24]=$SCR_GRP[1].$MCH_POS_Y;
2575: L P[2575] 800cm/min CNT100 COORD PTH ;
:SR[23]=$SCR_GRP[1].$MCH_POS_X;
:SR[24]=$SCR_GRP[1].$MCH_POS_Y;
2576: L P[2576] 800cm/min CNT100 COORD PTH ;
:SR[23]=$SCR_GRP[1].$MCH_POS_X;
:SR[24]=$SCR_GRP[1].$MCH_POS_Y;
2577: L P[2577] 800cm/min CNT100 COORD PTH ;
:SR[23]=$SCR_GRP[1].$MCH_POS_X;
:SR[24]=$SCR_GRP[1].$MCH_POS_Y;
2578: L P[2578] 800cm/min CNT100 COORD PTH ;
:SR[23]=$SCR_GRP[1].$MCH_POS_X;
:SR[24]=$SCR_GRP[1].$MCH_POS_Y;
2579: L P[2579] 800cm/min CNT100 COORD PTH ;
:SR[23]=$SCR_GRP[1].$MCH_POS_X;
:SR[24]=$SCR_GRP[1].$MCH_POS_Y;
2580: L P[2580] 800cm/min CNT100 COORD PTH ;
:SR[23]=$SCR_GRP[1].$MCH_POS_X;
:SR[24]=$SCR_GRP[1].$MCH_POS_Y;
2581: L P[2581] 800cm/min CNT100 COORD PTH ;
:SR[23]=$SCR_GRP[1].$MCH_POS_X;
:SR[24]=$SCR_GRP[1].$MCH_POS_Y;
2582: L P[2582] 800cm/min CNT100 COORD PTH ;
:SR[23]=$SCR_GRP[1].$MCH_POS_X;
:SR[24]=$SCR_GRP[1].$MCH_POS_Y;
2583: L P[2583] 800cm/min CNT100 COORD PTH ;
:SR[23]=$SCR_GRP[1].$MCH_POS_X;
:SR[24]=$SCR_GRP[1].$MCH_POS_Y;
2584: L P[2584] 800cm/min CNT100 COORD PTH ;
:SR[23]=$SCR_GRP[1].$MCH_POS_X;
:SR[24]=$SCR_GRP[1].$MCH_POS_Y;
2585: L P[2585] 800cm/min CNT100 COORD PTH ;
:SR[23]=$SCR_GRP[1].$MCH_POS_X;
:SR[24]=$SCR_GRP[1].$MCH_POS_Y;
2586: L P[2586] 800cm/min CNT100 COORD PTH ;
:SR[23]=$SCR_GRP[1].$MCH_POS_X;
:SR[24]=$SCR_GRP[1].$MCH_POS_Y;
2587: L P[2587] 800cm/min CNT100 COORD PTH ;
:SR[23]=$SCR_GRP[1].$MCH_POS_X;
:SR[24]=$SCR_GRP[1].$MCH_POS_Y;
2588: L P[2588] 800cm/min CNT100 COORD PTH ;
:SR[23]=$SCR_GRP[1].$MCH_POS_X;
:SR[24]=$SCR_GRP[1].$MCH_POS_Y;
2589: L P[2589] 800cm/min CNT100 COORD PTH ;
:SR[23]=$SCR_GRP[1].$MCH_POS_X;
:SR[24]=$SCR_GRP[1].$MCH_POS_Y;
2590: L P[2590] 800cm/min CNT100 COORD PTH ;
:SR[23]=$SCR_GRP[1].$MCH_POS_X;
:SR[24]=$SCR_GRP[1].$MCH_POS_Y;
2591: L P[2591] 800cm/min CNT100 COORD PTH ;
:SR[23]=$SCR_GRP[1].$MCH_POS_X;
:SR[24]=$SCR_GRP[1].$MCH_POS_Y;
2592: L P[2592] 800cm/min CNT100 COORD PTH ;
:SR[23]=$SCR_GRP[1].$MCH_POS_X;
:SR[24]=$SCR_GRP[1].$MCH_POS_Y;
2593: L P[2593] 800cm/min CNT100 COORD PTH ;
:SR[23]=$SCR_GRP[1].$MCH_POS_X;
:SR[24]=$SCR_GRP[1].$MCH_POS_Y;
2594: L P[2594] 800cm/min CNT100 COORD PTH ;
:SR[23]=$SCR_GRP[1].$MCH_POS_X;
:SR[24]=$SCR_GRP[1].$MCH_POS_Y;
2595: L P[2595] 800cm/min CNT100 COORD PTH ;
:SR[23]=$SCR_GRP[1].$MCH_POS_X;
:SR[24]=$SCR_GRP[1].$MCH_POS_Y;
2596: L P[2596] 800cm/min CNT100 COORD PTH ;
:SR[23]=$SCR_GRP[1].$MCH_POS_X;
:SR[24]=$SCR_GRP[1].$MCH_POS_Y;
2597: L P[2597] 800cm/min CNT100 COORD PTH ;
:SR[23]=$SCR_GRP[1].$MCH_POS_X;
:SR[24]=$SCR_GRP[1].$MCH_POS_Y;
2598: L P[2598] 800cm/min CNT100 COORD PTH ;
:SR[23]=$SCR_GRP[1].$MCH_POS_X;
:SR[24]=$SCR_GRP[1].$MCH_POS_Y;
2599: L P[2599] 800cm/min CNT100 COORD PTH ;
:SR[23]=$SCR_GRP[1].$MCH_POS_X;
:SR[24]=$SCR_GRP[1].$MCH_POS_Y;
2600: L P[2600] 800cm/min CNT100 COORD PTH ;
:SR[23]=$SCR_GRP[1].$MCH_POS_X;
:SR[24]=$SCR_GRP[1].$MCH_POS_Y;
2601: L P[2601] 800cm/min CNT100 COORD PTH ;
:SR[23]=$SCR_GRP[1].$MCH_POS_X;
:SR[24]=$SCR_GRP[1].$MCH_POS_Y;
2602: L P[2602] 800cm/min CNT100 COORD PTH ;
:SR[23]=$SCR_GRP[1].$MCH_POS_X;
:SR[24]=$SCR_GRP[1].$MCH_POS_Y;
2603: L P[2603] 800cm/min CNT100 COORD PTH ;
:SR[23]=$SCR_GRP[1].$MCH_POS_X;
:SR[24]=$SCR_GRP[1].$MCH_POS_Y;
2604: L P[2604] 800cm/min CNT100 COORD PTH ;
:SR[23]=$SCR_GRP[1].$MCH_POS_X;
:SR[24]=$SCR_GRP[1].$MCH_POS_Y;
2605: L P[2605] 800cm/min CNT100 COORD PTH ;
:SR[23]=$SCR_GRP[1].$MCH_POS_X;
:SR[24]=$SCR_GRP[1].$MCH_POS_Y;
2606: L P[2606] 800cm/min CNT100 COORD PTH ;
:SR[23]=$SCR_GRP[1].$MCH_POS_X;
:SR[24]=$SCR_GRP[1].$MCH_POS_Y;
2607: L P[2607] 800cm/min CNT100 COORD PTH ;
:SR[23]=$SCR_GRP[1].$MCH_POS_X;
:SR[24]=$SCR_GRP[1].$MCH_POS_Y;
2608: L P[2608] 800cm/min CNT100 COORD PTH ;
:SR[23]=$SCR_GRP[1].$MCH_POS_X;
:SR[24]=$SCR_GRP[1].$MCH_POS_Y;
2609: L P[2609] 800cm/min CNT100 COORD PTH ;
:SR[23]=$SCR_GRP[1].$MCH_POS_X;
:SR[24]=$SCR_GRP[1].$MCH_POS_Y;
2610: L P[2610] 800cm/min CNT100 COORD PTH ;
:SR[23]=$SCR_GRP[1].$MCH_POS_X;
:SR[24]=$SCR_GRP[1].$MCH_POS_Y;
2611: L P[2611] 800cm/min CNT100 COORD PTH ;
:SR[23]=$SCR_GRP[1].$MCH_POS_X;
:SR[24]=$SCR_GRP[1].$MCH_POS_Y;
2612: L P[2612] 800cm/min CNT100 COORD PTH ;
:SR[23]=$SCR_GRP[1].$MCH_POS_X;
:SR[24]=$SCR_GRP[1].$MCH_POS_Y;
2613: L P[2613] 800cm/min CNT100 COORD PTH ;
:SR[23]=$SCR_GRP[1].$MCH_POS_X;
:SR[24]=$SCR_GRP[1].$MCH_POS_Y;
2614: L P[2614] 800cm/min CNT100 COORD PTH ;
:SR[23]=$SCR_GRP[1].$MCH_POS_X;
:SR[24]=$SCR_GRP[1].$MCH_POS_Y;
2615: L P[2615] 800cm/min CNT100 COORD PTH ;
:SR[23]=$SCR_GRP[1].$MCH_POS_X;
:SR[24]=$SCR_GRP[1].$MCH_POS_Y;
2616: L P[2616] 800cm/min CNT100 COORD PTH ;
:SR[23]=$SCR_GRP[1].$MCH_POS_X;
:SR[24]=$SCR_GRP[1].$MCH_POS_Y;
2617: L P[2617] 800cm/min CNT100 COORD PTH ;
:SR[23]=$SCR_GRP[1].$MCH_POS_X;
:SR[24]=$SCR_GRP[1].$MCH_POS_Y;
2618: L P[2618] 800cm/min CNT100 COORD PTH ;
:SR[23]=$SCR_GRP[1].$MCH_POS_X;
:SR[24]=$SCR_GRP[1].$MCH_POS_Y;
2619: L P[2619] 800cm/min CNT100 COORD PTH ;
:SR[23]=$SCR_GRP[1].$MCH_POS_X;
:SR[24]=$SCR_GRP[1].$MCH_POS_Y;
2620: L P[2620] 800cm/min CNT100 COORD PTH ;
:SR[23]=$SCR_GRP[1].$MCH_POS_X;
:SR[24]=$SCR_GRP[1].$MCH_POS_Y;
2621: L P[2621] 800cm/min CNT100 COORD PTH ;
:SR[23]=$SCR_GRP[1].$MCH_POS_X;
:SR[24]=$SCR_GRP[1].$MCH_POS_Y;
2622: L P[2622] 800cm/min CNT100 COORD PTH ;
:SR[23]=$SCR_GRP[1].$MCH_POS_X;
:SR[24]=$SCR_GRP[1].$MCH_POS_Y;
2623: L P[2623] 800cm/min CNT100 COORD PTH ;
:SR[23]=$SCR_GRP[1].$MCH_POS_X;
:SR[24]=$SCR_GRP[1].$MCH_POS_Y;
2624: L P[2624] 800cm/min CNT100 COORD PTH ;
:SR[23]=$SCR_GRP[1].$MCH_POS_X;
:SR[24]=$SCR_GRP[1].$MCH_POS_Y;
2625: L P[2625] 800cm/min CNT100 COORD PTH ;
:SR[23]=$SCR_GRP[1].$MCH_POS_X;
:SR[24]=$SCR_GRP[1].$MCH_POS_Y;
2626: L P[2626] 800cm/min CNT100 COORD PTH ;
:SR[23]=$SCR_GRP[1].$MCH_POS_X;
:SR[24]=$SCR_GRP[1].$MCH_POS_Y;
2627: L P[2627] 800cm/min CNT100 COORD PTH ;
:SR[23]=$SCR_GRP[1].$MCH_POS_X;
:SR[24]=$SCR_GRP[1].$MCH_POS_Y;
2628: L P[2628] 800cm/min CNT100 COORD PTH ;
:SR[23]=$SCR_GRP[1].$MCH_POS_X;
:SR[24]=$SCR_GRP[1].$MCH_POS_Y;
2629: L P[2629] 800cm/min CNT100 COORD PTH ;
:SR[23]=$SCR_GRP[1].$MCH_POS_X;
:SR[24]=$SCR_GRP[1].$MCH_POS_Y;
2630: L P[2630] 800cm/min CNT100 COORD PTH ;
:SR[23]=$SCR_GRP[1].$MCH_POS_X;
:SR[24]=$SCR_GRP[1].$MCH_POS_Y;
2631: L P[2631] 800cm/min CNT100 COORD PTH ;
:SR[23]=$SCR_GRP[1].$MCH_POS_X;
:SR[24]=$SCR_GRP[1].$MCH_POS_Y;
2632: L P[2632] 800cm/min CNT100 COORD PTH ;
:SR[23]=$SCR_GRP[1].$MCH_POS_X;
:SR[24]=$SCR_GRP[1].$MCH_POS_Y;
2633: L P[2633] 800cm/min CNT100 COORD PTH ;
:SR[23]=$SCR_GRP[1].$MCH_POS_X;
:SR[24]=$SCR_GRP[1].$MCH_POS_Y;
2634: L P[2634] 800cm/min CNT100 COORD PTH ;
:SR[23]=$SCR_GRP[1].$MCH_POS_X;
:SR[24]=$SCR_GRP[1].$MCH_POS_Y;
2635: L P[2635] 800cm/min CNT100 COORD PTH ;
:SR[23]=$SCR_GRP[1].$MCH_POS_X;
:SR[24]=$SCR_GRP[1].$MCH_POS_Y;
2636: L P[2636] 800cm/min CNT100 COORD PTH ;
:SR[23]=$SCR_GRP[1].$MCH_POS_X;
:SR[24]=$SCR_GRP[1].$MCH_POS_Y;
2637: L P[2637] 800cm/min CNT100 COORD PTH ;
:SR[23]=$SCR_GRP[1].$MCH_POS_X;
:SR[24]=$SCR_GRP[1].$MCH_POS_Y;
2638: L P[2638] 800cm/min CNT100 COORD PTH ;
:SR[23]=$SCR_GRP[1].$MCH_POS_X;
:SR[24]=$SCR_GRP[1].$MCH_POS_Y;
2639: L P[2639] 800cm/min CNT100 COORD PTH ;
:SR[23]=$SCR_GRP[1].$MCH_POS_X;
:SR[24]=$SCR_GRP[1].$MCH_POS_Y;
2640: L P[2640] 800cm/min CNT100 COORD PTH ;
:SR[23]=$SCR_GRP[1].$MCH_POS_X;
:SR[24]=$SCR_GRP[1].$MCH_POS_Y;
2641: L P[2641] 800cm/min CNT100 COORD PTH ;
:SR[23]=$SCR_GRP[1].$MCH_POS_X;
:SR[24]=$SCR_GRP[1].$MCH_POS_Y;
2642: L P[2642] 800cm/min CNT100 COORD PTH ;
:SR[23]=$SCR_GRP[1].$MCH_POS_X;
:SR[24]=$SCR_GRP[1].$MCH_POS_Y;
2643: L P[2643] 800cm/min CNT100 COORD PTH ;
:SR[23]=$SCR_GRP[1].$MCH_POS_X;
:SR[24]=$SCR_GRP[1].$MCH_POS_Y;
2644: L P[2644] 800cm/min CNT100 COORD PTH ;
:SR[23]=$SCR_GRP[1].$MCH_POS_X;
:SR[24]=$SCR_GRP[1].$MCH_POS_Y;
2645: L P[2645] 800cm/min CNT100 COORD PTH ;
:SR[23]=$SCR_GRP[1].$MCH_POS_X;
:SR[24]=$SCR_GRP[1].$MCH_POS_Y;
2646: L P[2646] 800cm/min CNT100 COORD PTH ;
:SR[23]=$SCR_GRP[1].$MCH_POS_X;
:SR[24]=$SCR_GRP[1].$MCH_POS_Y;
2647: L P[2647] 800cm/min CNT100 COORD PTH ;
:SR[23]=$SCR_GRP[1].$MCH_POS_X;
:SR[24]=$SCR_GRP[1].$MCH_POS_Y;
2648: L P[2648] 800cm/min CNT100 COORD PTH ;
:SR[23]=$SCR_GRP[1].$MCH_POS_X;
:SR[24]=$SCR_GRP[1].$MCH_POS_Y;
2649: L P[2649] 800cm/min CNT100 COORD PTH ;
:SR[23]=$SCR_GRP[1].$MCH_POS_X;
:SR[24]=$SCR_GRP[1].$MCH_POS_Y;
2650: L P[2650] 800cm/min CNT100 COORD PTH ;
:SR[23]=$SCR_GRP[1].$MCH_POS_X;
:SR[24]=$SCR_GRP[1].$MCH_POS_Y;
2651: L P[2651] 800cm/min CNT100 COORD PTH ;
:SR[23]=$SCR_GRP[1].$MCH_POS_X;
:SR[24]=$SCR_GRP[1].$MCH_POS_Y;
2652: L P[2652] 800cm/min CNT100 COORD PTH ;
:SR[23]=$SCR_GRP[1].$MCH_POS_X;
:SR[24]=$SCR_GRP[1].$MCH_POS_Y;
2653: L P[2653] 800cm/min CNT100 COORD PTH ;
:SR[23]=$SCR_GRP[1].$MCH_POS_X;
:SR[24]=$SCR_GRP[1].$MCH_POS_Y;
2654: L P[2654] 800cm/min CNT100 COORD PTH ;
:SR[23]=$SCR_GRP[1].$MCH_POS_X;
:SR[24]=$SCR_GRP[1].$MCH_POS_Y;
2655: L P[2655] 800cm/min CNT100 COORD PTH ;
:SR[23]=$SCR_GRP[1].$MCH_POS_X;
:SR[24]=$SCR_GRP[1].$MCH_POS_Y;
2656: L P[2656] 800cm/min CNT100 COORD PTH ;
:SR[23]=$SCR_GRP[1].$MCH_POS_X;
:SR[24]=$SCR_GRP[1].$MCH_POS_Y;
2657: L P[2657] 800cm/min CNT100 COORD PTH ;
:SR[23]=$SCR_GRP[1].$MCH_POS_X;
:SR[24]=$SCR_GRP[1].$MCH_POS_Y;
2658: L P[2658] 800cm/min CNT100 COORD PTH ;
:SR[23]=$SCR_GRP[1].$MCH_POS_X;
:SR[24]=$SCR_GRP[1].$MCH_POS_Y;
2659: L P[2659] 800cm/min CNT100 COORD PTH ;
:SR[23]=$SCR_GRP[1].$MCH_POS_X;
:SR[24]=$SCR_GRP[1].$MCH_POS_Y;
2660: L P[2660] 800cm/min CNT100 COORD PTH ;
:SR[23]=$SCR_GRP[1].$MCH_POS_X;
:SR[24]=$SCR_GRP[1].$MCH_POS_Y;
2661: L P[2661] 800cm/min CNT100 COORD PTH ;
:SR[23]=$SCR_GRP[1].$MCH_POS_X;
:SR[24]=$SCR_GRP[1].$MCH_POS_Y;
2662: L P[2662] 800cm/min CNT100 COORD PTH ;
:SR[23]=$SCR_GRP[1].$MCH_POS_X;
:SR[24]=$SCR_GRP[1].$MCH_POS_Y;
2663: L P[2663] 800cm/min CNT100 COORD PTH ;
:SR[23]=$SCR_GRP[1].$MCH_POS_X;
:SR[24]=$SCR_GRP[1].$MCH_POS_Y;
2664: L P[2664] 800cm/min CNT100 COORD PTH ;
:SR[23]=$SCR_GRP[1].$MCH_POS_X;
:SR[24]=$SCR_GRP[1].$MCH_POS_Y;
2665: L P[2665] 800cm/min CNT100 COORD PTH ;
:SR[23]=$SCR_GRP[1].$MCH_POS_X;
:SR[24]=$SCR_GRP[1].$MCH_POS_Y;
2666: L P[2666] 800cm/min CNT100 COORD PTH ;
:SR[23]=$SCR_GRP[1].$MCH_POS_X;
:SR[24]=$SCR_GRP[1].$MCH_POS_Y;
2667: L P[2667] 800cm/min CNT100 COORD PTH ;
:SR[23]=$SCR_GRP[1].$MCH_POS_X;
:SR[24]=$SCR_GRP[1].$MCH_POS_Y;
2668: L P[2668] 800cm/min CNT100 COORD PTH ;
:SR[23]=$SCR_GRP[1].$MCH_POS_X;
:SR[24]=$SCR_GRP[1].$MCH_POS_Y;
2669: L P[2669] 800cm/min CNT100 COORD PTH ;
:SR[23]=$SCR_GRP[1].$MCH_POS_X;
:SR[24]=$SCR_GRP[1].$MCH_POS_Y;
2670: L P[2670] 800cm/min CNT100 COORD PTH ;
:SR[23]=$SCR_GRP[1].$MCH_POS_X;
:SR[24]=$SCR_GRP[1].$MCH_POS_Y;
2671: L P[2671] 800cm/min CNT100 COORD PTH ;
:SR[23]=$SCR_GRP[1].$MCH_POS_X;
:SR[24]=$SCR_GRP[1].$MCH_POS_Y;
2672: L P[2672] 800cm/min CNT100 COORD PTH ;
:SR[23]=$SCR_GRP[1].$MCH_POS_X;
:SR[24]=$SCR_GRP[1].$MCH_POS_Y;
2673: L P[2673] 800cm/min CNT100 COORD PTH ;
:SR[23]=$SCR_GRP[1].$MCH_POS_X;
:SR[24]=$SCR_GRP[1].$MCH_POS_Y;
2674: L P[2674] 800cm/min CNT100 COORD PTH ;
:SR[23]=$SCR_GRP[1].$MCH_POS_X;
:SR[24]=$SCR_GRP[1].$MCH_POS_Y;
2675: L P[2675] 800cm/min CNT100 COORD PTH ;
:SR[23]=$SCR_GRP[1].$MCH_POS_X;
:SR[24]=$SCR_GRP[1].$MCH_POS_Y;
2676: L P[2676] 800cm/min CNT100 COORD PTH ;
:SR[23]=$SCR_GRP[1].$MCH_POS_X;
:SR[24]=$SCR_GRP[1].$MCH_POS_Y;
2677: L P[2677] 800cm/min CNT100 COORD PTH ;
:SR[23]=$SCR_GRP[1].$MCH_POS_X;
:SR[24]=$SCR_GRP[1].$MCH_POS_Y;
2678: L P[2678] 800cm/min CNT100 COORD PTH ;
:SR[23]=$SCR_GRP[1].$MCH_POS_X;
:SR[24]=$SCR_GRP[1].$MCH_POS_Y;
2679: L P[2679] 800cm/min CNT100 COORD PTH ;
:SR[23]=$SCR_GRP[1].$MCH_POS_X;
:SR[24]=$SCR_GRP[1].$MCH_POS_Y;
2680: L P[2680] 800cm/min CNT100 COORD PTH ;
:SR[23]=$SCR_GRP[1].$MCH_POS_X;
:SR[24]=$SCR_GRP[1].$MCH_POS_Y;
2681: L P[2681] 800cm/min CNT100 COORD PTH ;
:SR[23]=$SCR_GRP[1].$MCH_POS_X;
:SR[24]=$SCR_GRP[1].$MCH_POS_Y;
2682: L P[2682] 800cm/min CNT100 COORD PTH ;
:SR[23]=$SCR_GRP[1].$MCH_POS_X;
:SR[24]=$SCR_GRP[1].$MCH_POS_Y;
2683: L P[2683] 800cm/min CNT100 COORD PTH ;
:SR[23]=$SCR_GRP[1].$MCH_POS_X;
:SR[24]=$SCR_GRP[1].$MCH_POS_Y;
2684: L P[2684] 800cm/min CNT100 COORD PTH ;
:SR[23]=$SCR_GRP[1].$MCH_POS_X;
:SR[24]=$SCR_GRP[1].$MCH_POS_Y;
2685: L P[2685] 800cm/min CNT100 COORD PTH ;
:SR[23]=$SCR_GRP[1].$MCH_POS_X;
:SR[24]=$SCR_GRP[1].$MCH_POS_Y;
2686: L P[2686] 800cm/min CNT100 COORD PTH ;
:SR[23]=$SCR_GRP[1].$MCH_POS_X;
:SR[24]=$SCR_GRP[1].$MCH_POS_Y;
2687: L P[2687] 800cm/min CNT100 COORD PTH ;
:SR[23]=$SCR_GRP[1].$MCH_POS_X;
:SR[24]=$SCR_GRP[1].$MCH_POS_Y;
2688: L P[2688] 800cm/min CNT100 COORD PTH ;
:SR[23]=$SCR_GRP[1].$MCH_POS_X;
:SR[24]=$SCR_GRP[1].$MCH_POS_Y;
2689: L P[2689] 800cm/min CNT100 COORD PTH ;
:SR[23]=$SCR_GRP[1].$MCH_POS_X;
:SR[24]=$SCR_GRP[1].$MCH_POS_Y;
2690: L P[2690] 800cm/min CNT100 COORD PTH ;
:SR[23]=$SCR_GRP[1].$MCH_POS_X;
:SR[24]=$SCR_GRP[1].$MCH_POS_Y;
2691: L P[2691] 800cm/min CNT100 COORD PTH ;
:SR[23]=$SCR_GRP[1].$MCH_POS_X;
:SR[24]=$SCR_GRP[1].$MCH_POS_Y;
2692: L P[2692] 800cm/min CNT100 COORD PTH ;
:SR[23]=$SCR_GRP[1].$MCH_POS_X;
:SR[24]=$SCR_GRP[1].$MCH_POS_Y;
2693: L P[2693] 800cm/min CNT100 COORD PTH ;
:SR[23]=$SCR_GRP[1].$MCH_POS_X;
:SR[24]=$SCR_GRP[1].$MCH_POS_Y;
2694: L P[2694] 800cm/min CNT100 COORD PTH ;
:SR[23]=$SCR_GRP[1].$MCH_POS_X;
:SR[24]=$SCR_GRP[1].$MCH_POS_Y;
2695: L P[2695] 800cm/min CNT100 COORD PTH ;
:SR[23]=$SCR_GRP[1].$MCH_POS_X;
:SR[24]=$SCR_GRP[1].$MCH_POS_Y;
2696: L P[2696] 800cm/min CNT100 COORD PTH ;
:SR[23]=$SCR_GRP[1].$MCH_POS_X;
:SR[24]=$SCR_GRP[1].$MCH_POS_Y;
2697: L P[2697] 800cm/min CNT100 COORD PTH ;
:SR[23]=$SCR_GRP[1].$MCH_POS_X;
:SR[24]=$SCR_GRP[1].$MCH_POS_Y;
2698: L P[2698] 800cm/min CNT100 COORD PTH ;
:SR[23]=$SCR_GRP[1].$MCH_POS_X;
:SR[24]=$SCR_GRP[1].$MCH_POS_Y;
2699: L P[2699] 800cm/min CNT100 COORD PTH ;
:SR[23]=$SCR_GRP[1].$MCH_POS_X;
:SR[24]=$SCR_GRP[1].$MCH_POS_Y;
2700: L P[2700] 800cm/min CNT100 COORD PTH ;
:SR[23]=$SCR_GRP[1].$MCH_POS_X;
:SR[24]=$SCR_GRP[1].$MCH_POS_Y;
2701: L P[2701] 800cm/min CNT100 COORD PTH ;
:SR[23]=$SCR_GRP[1].$MCH_POS_X;
:SR[24]=$SCR_GRP[1].$MCH_POS_Y;
2702: L P[2702] 800cm/min CNT100 COORD PTH ;
:SR[23]=$SCR_GRP[1].$MCH_POS_X;
:SR[24]=$SCR_GRP[1].$MCH_POS_Y;
2703: L P[2703] 800cm/min CNT100 COORD PTH ;
:SR[23]=$SCR_GRP[1].$MCH_POS_X;
:SR[24]=$SCR_GRP[1].$MCH_POS_Y;
2704: L P[2704] 800cm/min CNT100 COORD PTH ;
:SR[23]=$SCR_GRP[1].$MCH_POS_X;
:SR[24]=$SCR_GRP[1].$MCH_POS_Y;
2705: L P[2705] 800cm/min CNT100 COORD PTH ;
:SR[23]=$SCR_GRP[1].$MCH_POS_X;
:SR[24]=$SCR_GRP[1].$MCH_POS_Y;
2706: L P[2706] 800cm/min CNT100 COORD PTH ;
:SR[23]=$SCR_GRP[1].$MCH_POS_X;
:SR[24]=$SCR_GRP[1].$MCH_POS_Y;
2707: L P[2707] 800cm/min CNT100 COORD PTH ;
:SR[23]=$SCR_GRP[1].$MCH_POS_X;
:SR[24]=$SCR_GRP[1].$MCH_POS_Y;
2708: L P[2708] 800cm/min CNT100 COORD PTH ;
:SR[23]=$SCR_GRP[1].$MCH_POS_X;
:SR[24]=$SCR_GRP[1].$MCH_POS_Y;
2709: L P[2709] 800cm/min CNT100 COORD PTH ;
:SR[23]=$SCR_GRP[1].$MCH_POS_X;
:SR[24]=$SCR_GRP[1].$MCH_POS_Y;
2710: L P[2710] 800cm/min CNT100 COORD PTH ;
:SR[23]=$SCR_GRP[1].$MCH_POS_X;
:SR[24]=$SCR_GRP[1].$MCH_POS_Y;
2711: L P[2711] 800cm/min CNT100 COORD PTH ;
:SR[23]=$SCR_GRP[1].$MCH_POS_X;
:SR[24]=$SCR_GRP[1].$MCH_POS_Y;
2712: L P[2712] 800cm/min CNT100 COORD PTH ;
:SR[23]=$SCR_GRP[1].$MCH_POS_X;
:SR[24]=$SCR_GRP[1].$MCH_POS_Y;
2713: L P[2713] 800cm/min CNT100 COORD PTH ;
:SR[23]=$SCR_GRP[1].$MCH_POS_X;
:SR[24]=$SCR_GRP[1].$MCH_POS_Y;
2714: L P[2714] 800cm/min CNT100 COORD PTH ;
:SR[23]=$SCR_GRP[1].$MCH_POS_X;
:SR[24]=$SCR_GRP[1].$MCH_POS_Y;
2715: L P[2715] 800cm/min CNT100 COORD PTH ;
:SR[23]=$SCR_GRP[1].$MCH_POS_X;
:SR[24]=$SCR_GRP[1].$MCH_POS_Y;
2716: L P[2716] 800cm/min CNT100 COORD PTH ;
:SR[23]=$SCR_GRP[1].$MCH_POS_X;
:SR[24]=$SCR_GRP[1].$MCH_POS_Y;
2717: L P[2717] 800cm/min CNT100 COORD PTH ;
:SR[23]=$SCR_GRP[1].$MCH_POS_X;
:SR[24]=$SCR_GRP[1].$MCH_POS_Y;
2718: L P[2718] 800cm/min CNT100 COORD PTH ;
:SR[23]=$SCR_GRP[1].$MCH_POS_X;
:SR[24]=$SCR_GRP[1].$MCH_POS_Y;
2719: L P[2719] 800cm/min CNT100 COORD PTH ;
:SR[23]=$SCR_GRP[1].$MCH_POS_X;
:SR[24]=$SCR_GRP[1].$MCH_POS_Y;
2720: L P[2720] 800cm/min CNT100 COORD PTH ;
:SR[23]=$SCR_GRP[1].$MCH_POS_X;
:SR[24]=$SCR_GRP[1].$MCH_POS_Y;
2721: L P[2721] 800cm/min CNT100 COORD PTH ;
:SR[23]=$SCR_GRP[1].$MCH_POS_X;
:SR[24]=$SCR_GRP[1].$MCH_POS_Y;
2722: L P[2722] 800cm/min CNT100 COORD PTH ;
:SR[23]=$SCR_GRP[1].$MCH_POS_X;
:SR[24]=$SCR_GRP[1].$MCH_POS_Y;
2723: L P[2723] 800cm/min CNT100 COORD PTH ;
:SR[23]=$SCR_GRP[1].$MCH_POS_X;
:SR[24]=$SCR_GRP[1].$MCH_POS_Y;
2724: L P[2724] 800cm/min CNT100 COORD PTH ;
:SR[23]=$SCR_GRP[1].$MCH_POS_X;
:SR[24]=$SCR_GRP[1].$MCH_POS_Y;
2725: L P[2725] 800cm/min CNT100 COORD PTH ;
:SR[23]=$SCR_GRP[1].$MCH_POS_X;
:SR[24]=$SCR_GRP[1].$MCH_POS_Y;
2726: L P[2726] 800cm/min CNT100 COORD PTH ;
:SR[23]=$SCR_GRP[1].$MCH_POS_X;
:SR[24]=$SCR_GRP[1].$MCH_POS_Y;
2727: L P[2727] 800cm/min CNT100 COORD PTH ;
:SR[23]=$SCR_GRP[1].$MCH_POS_X;
:SR[24]=$SCR_GRP[1].$MCH_POS_Y;
2728: L P[2728] 800cm/min CNT100 COORD PTH ;
:SR[23]=$SCR_GRP[1].$MCH_POS_X;
:SR[24]=$SCR_GRP[1].$MCH_POS_Y;
2729: L P[2729] 800cm/min CNT100 COORD PTH ;
:SR[23]=$SCR_GRP[1].$MCH_POS_X;
:SR[24]=$SCR_GRP[1].$MCH_POS_Y;
2730: L P[2730] 800cm/min CNT100 COORD PTH ;
:SR[23]=$SCR_GRP[1].$MCH_POS_X;
:SR[24]=$SCR_GRP[1].$MCH_POS_Y;
2731: L P[2731] 800cm/min CNT100 COORD PTH ;
:SR[23]=$SCR_GRP[1].$MCH_POS_X;
:SR[24]=$SCR_GRP[1].$MCH_POS_Y;
2732: L P[2732] 800cm/min CNT100 COORD PTH ;
:SR[23]=$SCR_GRP[1].$MCH_POS_X;
:SR[24]=$SCR_GRP[1].$MCH_POS_Y;
2733: L P[2733] 800cm/min CNT100 COORD PTH ;
:SR[23]=$SCR_GRP[1].$MCH_POS_X;
:SR[24]=$SCR_GRP[1].$MCH_POS_Y;
2734: L P[2734] 800cm/min CNT100 COORD PTH ;
:SR[23]=$SCR_GRP[1].$MCH_POS_X;
:SR[24]=$SCR_GRP[1].$MCH_POS_Y;
2735: L P[2735] 800cm/min CNT100 COORD PTH ;
:SR[23]=$SCR_GRP[1].$MCH_POS_X;
:SR[24]=$SCR_GRP[1].$MCH_POS_Y;
2736: L P[2736] 800cm/min CNT100 COORD PTH ;
:SR[23]=$SCR_GRP[1].$MCH_POS_X;
:SR[24]=$SCR_GRP[1].$MCH_POS_Y;
2737: L P[2737] 800cm/min CNT100 COORD PTH ;
:SR[23]=$SCR_GRP[1].$MCH_POS_X;
:SR[24]=$SCR_GRP[1].$MCH_POS_Y;
2738: L P[2738] 800cm/min CNT100 COORD PTH ;
:SR[23]=$SCR_GRP[1].$MCH_POS_X;
:SR[24]=$SCR_GRP[1].$MCH_POS_Y;
2739: L P[2739] 800cm/min CNT100 COORD PTH ;
:SR[23]=$SCR_GRP[1].$MCH_POS_X;
:SR[24]=$SCR_GRP[1].$MCH_POS_Y;
2740: L P[2740] 800cm/min CNT100 COORD PTH ;
:SR[23]=$SCR_GRP[1].$MCH_POS_X;
:SR[24]=$SCR_GRP[1].$MCH_POS_Y;
2741: L P[2741] 800cm/min CNT100 COORD PTH ;
:SR[23]=$SCR_GRP[1].$MCH_POS_X;
:SR[24]=$SCR_GRP[1].$MCH_POS_Y;
2742: L P[2742] 800cm/min CNT100 COORD PTH ;
:SR[23]=$SCR_GRP[1].$MCH_POS_X;
:SR[24]=$SCR_GRP[1].$MCH_POS_Y;
2743: L P[2743] 800cm/min CNT100 COORD PTH ;
:SR[23]=$SCR_GRP[1].$MCH_POS_X;
:SR[24]=$SCR_GRP[1].$MCH_POS_Y;
2744: L P[2744] 800cm/min CNT100 COORD PTH ;
:SR[23]=$SCR_GRP[1].$MCH_POS_X;
:SR[24]=$SCR_GRP[1].$MCH_POS_Y;
2745: L P[2745] 800cm/min CNT100 COORD PTH ;
:SR[23]=$SCR_GRP[1].$MCH_POS_X;
:SR[24]=$SCR_GRP[1].$MCH_POS_Y;
2746: L P[2746] 800cm/min CNT100 COORD PTH ;
:SR[23]=$SCR_GRP[1].$MCH_POS_X;
:SR[24]=$SCR_GRP[1].$MCH_POS_Y;
2747: L P[2747] 800cm/min CNT100 COORD PTH ;
:SR[23]=$SCR_GRP[1].$MCH_POS_X;
:SR[24]=$SCR_GRP[1].$MCH_POS_Y;
2748: L P[2748] 800cm/min CNT100 COORD PTH ;
:SR[23]=$SCR_GRP[1].$MCH_POS_X;
:SR[24]=$SCR_GRP[1].$MCH_POS_Y;
2749: L P[2749] 800cm/min CNT100 COORD PTH ;
:SR[23]=$SCR_GRP[1].$MCH_POS_X;
:SR[24]=$SCR_GRP[1].$MCH_POS_Y;
2750: L P[2750] 800cm/min CNT100 COORD PTH ;
:SR[23]=$SCR_GRP[1].$MCH_POS_X;
:SR[24]=$SCR_GRP[1].$MCH_POS_Y;
2751: L P[2751] 800cm/min CNT100 COORD PTH ;
:SR[23]=$SCR_GRP[1].$MCH_POS_X;
:SR[24]=$SCR_GRP[1].$MCH_POS_Y;
2752: L P[2752] 800cm/min CNT100 COORD PTH ;
:SR[23]=$SCR_GRP[1].$MCH_POS_X;
:SR[24]=$SCR_GRP[1].$MCH_POS_Y;
2753: L P[2753] 800cm/min CNT100 COORD PTH ;
:SR[23]=$SCR_GRP[1].$MCH_POS_X;
:SR[24]=$SCR_GRP[1].$MCH_POS_Y;
2754: L P[2754] 800cm/min CNT100 COORD PTH ;
:SR[23]=$SCR_GRP[1].$MCH_POS_X;
:SR[24]=$SCR_GRP[1].$MCH_POS_Y;
2755: L P[2755] 800cm/min CNT100 COORD PTH ;
:SR[23]=$SCR_GRP[1].$MCH_POS_X;
:SR[24]=$SCR_GRP[1].$MCH_POS_Y;
2756: L P[2756] 800cm/min CNT100 COORD PTH ;
:SR[23]=$SCR_GRP[1].$MCH_POS_X;
:SR[24]=$SCR_GRP[1].$MCH_POS_Y;
2757: L P[2757] 800cm/min CNT100 COORD PTH ;
:SR[23]=$SCR_GRP[1].$MCH_POS_X;
:SR[24]=$SCR_GRP[1].$MCH_POS_Y;
2758: L P[2758] 800cm/min CNT100 COORD PTH ;
:SR[23]=$SCR_GRP[1].$MCH_POS_X;
:SR[24]=$SCR_GRP[1].$MCH_POS_Y;
2759: L P[2759] 800cm/min CNT100 COORD PTH ;
:SR[23]=$SCR_GRP[1].$MCH_POS_X;
:SR[24]=$SCR_GRP[1].$MCH_POS_Y;
2760: L P[2760] 800cm/min CNT100 COORD PTH ;
:SR[23]=$SCR_GRP[1].$MCH_POS_X;
:SR[24]=$SCR_GRP[1].$MCH_POS_Y;
2761: L P[2761] 800cm/min CNT100 COORD PTH ;
:SR[23]=$SCR_GRP[1].$MCH_POS_X;
:SR[24]=$SCR_GRP[1].$MCH_POS_Y;
2762: L P[2762] 800cm/min CNT100 COORD PTH ;
:SR[23]=$SCR_GRP[1].$MCH_POS_X;
:SR[24]=$SCR_GRP[1].$MCH_POS_Y;
2763: L P[2763] 800cm/min CNT100 COORD PTH ;
:SR[23]=$SCR_GRP[1].$MCH_POS_X;
:SR[24]=$SCR_GRP[1].$MCH_POS_Y;
2764: L P[2764] 800cm/min CNT100 COORD PTH ;
:SR[23]=$SCR_GRP[1].$MCH_POS_X;
:SR[24]=$SCR_GRP[1].$MCH_POS_Y;
2765: L P[2765] 800cm/min CNT100 COORD PTH ;
:SR[23]=$SCR_GRP[1].$MCH_POS_X;
:SR[24]=$SCR_GRP[1].$MCH_POS_Y;
2766: L P[2766] 800cm/min CNT100 COORD PTH ;
:SR[23]=$SCR_GRP[1].$MCH_POS_X;
:SR[24]=$SCR_GRP[1].$MCH_POS_Y;
2767: L P[2767] 800cm/min CNT100 COORD PTH ;
:SR[23]=$SCR_GRP[1].$MCH_POS_X;
:SR[24]=$SCR_GRP[1].$MCH_POS_Y;
2768: L P[2768] 800cm/min CNT100 COORD PTH ;
:SR[23]=$SCR_GRP[1].$MCH_POS_X;
:SR[24]=$SCR_GRP[1].$MCH_POS_Y;
2769: L P[2769] 800cm/min CNT100 COORD PTH ;
:SR[23]=$SCR_GRP[1].$MCH_POS_X;
:SR[24]=$SCR_GRP[1].$MCH_POS_Y;
2770: L P[2770] 800cm/min CNT100 COORD PTH ;
:SR[23]=$SCR_GRP[1].$MCH_POS_X;
:SR[24]=$SCR_GRP[1].$MCH_POS_Y;
2771: L P[2771] 800cm/min CNT100 COORD PTH ;
:SR[23]=$SCR_GRP[1].$MCH_POS_X;
:SR[24]=$SCR_GRP[1].$MCH_POS_Y;
2772: L P[2772] 800cm/min CNT100 COORD PTH ;
:SR[23]=$SCR_GRP[1].$MCH_POS_X;
:SR[24]=$SCR_GRP[1].$MCH_POS_Y;
2773: L P[2773] 800cm/min CNT100 COORD PTH ;
:SR[23]=$SCR_GRP[1].$MCH_POS_X;
:SR[24]=$SCR_GRP[1].$MCH_POS_Y;
2774: L P[2774] 800cm/min CNT100 COORD PTH ;
:SR[23]=$SCR_GRP[1].$MCH_POS_X;
:SR[24]=$SCR_GRP[1].$MCH_POS_Y;
2775: L P[2775] 800cm/min CNT100 COORD PTH ;
:SR[23]=$SCR_GRP[1].$MCH_POS_X;
:SR[24]=$SCR_GRP[1].$MCH_POS_Y;
2776: L P[2776] 800cm/min CNT100 COORD PTH ;
:SR[23]=$SCR_GRP[1].$MCH_POS_X;
:SR[24]=$SCR_GRP[1].$MCH_POS_Y;
2777: L P[2777] 800cm/min CNT100 COORD PTH ;
:SR[23]=$SCR_GRP[1].$MCH_POS_X;
:SR[24]=$SCR_GRP[1].$MCH_POS_Y;
2778: L P[2778] 800cm/min CNT100 COORD PTH ;
:SR[23]=$SCR_GRP[1].$MCH_POS_X;
:SR[24]=$SCR_GRP[1].$MCH_POS_Y;
2779: L P[2779] 800cm/min CNT100 COORD PTH ;
:SR[23]=$SCR_GRP[1].$MCH_POS_X;
:SR[24]=$SCR_GRP[1].$MCH_POS_Y;
2780: L P[2780] 800cm/min CNT100 COORD PTH ;
:SR[23]=$SCR_GRP[1].$MCH_POS_X;
:SR[24]=$SCR_GRP[1].$MCH_POS_Y;
2781: L P[2781] 800cm/min CNT100 COORD PTH ;
:SR[23]=$SCR_GRP[1].$MCH_POS_X;
:SR[24]=$SCR_GRP[1].$MCH_POS_Y;
2782: L P[2782] 800cm/min CNT100 COORD PTH ;
:SR[23]=$SCR_GRP[1].$MCH_POS_X;
:SR[24]=$SCR_GRP[1].$MCH_POS_Y;
2783: L P[2783] 800cm/min CNT100 COORD PTH ;
:SR[23]=$SCR_GRP[1].$MCH_POS_X;
:SR[24]=$SCR_GRP[1].$MCH_POS_Y;
2784: L P[2784] 800cm/min CNT100 COORD PTH ;
:SR[23]=$SCR_GRP[1].$MCH_POS_X;
:SR[24]=$SCR_GRP[1].$MCH_POS_Y;
2785: L P[2785] 800cm/min CNT100 COORD PTH ;
:SR[23]=$SCR_GRP[1].$MCH_POS_X;
:SR[24]=$SCR_GRP[1].$MCH_POS_Y;
2786: L P[2786] 800cm/min CNT100 COORD PTH ;
:SR[23]=$SCR_GRP[1].$MCH_POS_X;
:SR[24]=$SCR_GRP[1].$MCH_POS_Y;
2787: L P[2787] 800cm/min CNT100 COORD PTH ;
:SR[23]=$SCR_GRP[1].$MCH_POS_X;
:SR[24]=$SCR_GRP[1].$MCH_POS_Y;
2788: L P[2788] 800cm/min CNT100 COORD PTH ;
:SR[23]=$SCR_GRP[1].$MCH_POS_X;
:SR[24]=$SCR_GRP[1].$MCH_POS_Y;
2789: L P[2789] 800cm/min CNT100 COORD PTH ;
:SR[23]=$SCR_GRP[1].$MCH_POS_X;
:SR[24]=$SCR_GRP[1].$MCH_POS_Y;
2790: L P[2790] 800cm/min CNT100 COORD PTH ;
:SR[23]=$SCR_GRP[1].$MCH_POS_X;
:SR[24]=$SCR_GRP[1].$MCH_POS_Y;
2791: L P[2791] 800cm/min CNT100 COORD PTH ;
:SR[23]=$SCR_GRP[1].$MCH_POS_X;
:SR[24]=$SCR_GRP[1].$MCH_POS_Y;
2792: L P[2792] 800cm/min CNT100 COORD PTH ;
:SR[23]=$SCR_GRP[1].$MCH_POS_X;
:SR[24]=$SCR_GRP[1].$MCH_POS_Y;
2793: L P[2793] 800cm/min CNT100 COORD PTH ;
:SR[23]=$SCR_GRP[1].$MCH_POS_X;
:SR[24]=$SCR_GRP[1].$MCH_POS_Y;
2794: L P[2794] 800cm/min CNT100 COORD PTH ;
:SR[23]=$SCR_GRP[1].$MCH_POS_X;
:SR[24]=$SCR_GRP[1].$MCH_POS_Y;
2795: L P[2795] 800cm/min CNT100 COORD PTH ;
:SR[23]=$SCR_GRP[1].$MCH_POS_X;
:SR[24]=$SCR_GRP[1].$MCH_POS_Y;
2796: L P[2796] 800cm/min CNT100 COORD PTH ;
:SR[23]=$SCR_GRP[1].$MCH_POS_X;
:SR[24]=$SCR_GRP[1].$MCH_POS_Y;
2797: L P[2797] 800cm/min CNT100 COORD PTH ;
:SR[23]=$SCR_GRP[1].$MCH_POS_X;
:SR[24]=$SCR_GRP[1].$MCH_POS_Y;
2798: L P[2798] 800cm/min CNT100 COORD PTH ;
:SR[23]=$SCR_GRP[1].$MCH_POS_X;
:SR[24]=$SCR_GRP[1].$MCH_POS_Y;
2799: L P[2799] 800cm/min CNT100 COORD PTH ;
:SR[23]=$SCR_GRP[1].$MCH_POS_X;
:SR[24]=$SCR_GRP[1].$MCH_POS_Y;
2800: L P[2800] 800cm/min CNT100 COORD PTH ;
:SR[23]=$SCR_GRP[1].$MCH_POS_X;
:SR[24]=$SCR_GRP[1].$MCH_POS_Y;
2801: L P[2801] 800cm/min CNT100 COORD PTH ;
:SR[23]=$SCR_GRP[1].$MCH_POS_X;
:SR[24]=$SCR_GRP[1].$MCH_POS_Y;
2802: L P[2802] 800cm/min CNT100 COORD PTH ;
:SR[23]=$SCR_GRP[1].$MCH_POS_X;
:SR[24]=$SCR_GRP[1].$MCH_POS_Y;
2803: L P[2803] 800cm/min CNT100 COORD PTH ;
:SR[23]=$SCR_GRP[1].$MCH_POS_X;
:SR[24]=$SCR_GRP[1].$MCH_POS_Y;
2804: L P[2804] 800cm/min CNT100 COORD PTH ;
:SR[23]=$SCR_GRP[1].$MCH_POS_X;
:SR[24]=$SCR_GRP[1].$MCH_POS_Y;
2805: L P[2805] 800cm/min CNT100 COORD PTH ;
:SR[23]=$SCR_GRP[1].$MCH_POS_X;
:SR[24]=$SCR_GRP[1].$MCH_POS_Y;
2806: L P[2806] 800cm/min CNT100 COORD PTH ;
:SR[23]=$SCR_GRP[1].$MCH_POS_X;
:SR[24]=$SCR_GRP[1].$MCH_POS_Y;
2807: L P[2807] 800cm/min CNT100 COORD PTH ;
:SR[23]=$SCR_GRP[1].$MCH_POS_X;
:SR[24]=$SCR_GRP[1].$MCH_POS_Y;
2808: L P[2808] 800cm/min CNT100 COORD PTH ;
:SR[23]=$SCR_GRP[1].$MCH_POS_X;
:SR[24]=$SCR_GRP[1].$MCH_POS_Y;
2809: L P[2809] 800cm/min CNT100 COORD PTH ;
:SR[23]=$SCR_GRP[1].$MCH_POS_X;
:SR[24]=$SCR_GRP[1].$MCH_POS_Y;
2810: L P[2810] 800cm/min CNT100 COORD PTH ;
:SR[23]=$SCR_GRP[1].$MCH_POS_X;
:SR[24]=$SCR_GRP[1].$MCH_POS_Y;
2811: L P[2811] 800cm/min CNT100 COORD PTH ;
:SR[23]=$SCR_GRP[1].$MCH_POS_X;
:SR[24]=$SCR_GRP[1].$MCH_POS_Y;
2812: L P[2812] 800cm/min CNT100 COORD PTH ;
:SR[23]=$SCR_GRP[1].$MCH_POS_X;
:SR[24]=$SCR_GRP[1].$MCH_POS_Y;
2813: L P[2813] 800cm/min CNT100 COORD PTH ;
:SR[23]=$SCR_GRP[1].$MCH_POS_X;
:SR[24]=$SCR_GRP[1].$MCH_POS_Y;
2814: L P[2814] 800cm/min CNT100 COORD PTH ;
:SR[23]=$SCR_GRP[1].$MCH_POS_X;
:SR[24]=$SCR_GRP[1].$MCH_POS_Y;
2815: L P[2815] 800cm/min CNT100 COORD PTH ;
:SR[23]=$SCR_GRP[1].$MCH_POS_X;
:SR[24]=$SCR_GRP[1].$MCH_POS_Y;
2816: L P[2816] 800cm/min CNT100 COORD PTH ;
:SR[23]=$SCR_GRP[1].$MCH_POS_X;
:SR[24]=$SCR_GRP[1].$MCH_POS_Y;
2817: L P[2817] 800cm/min CNT100 COORD PTH ;
:SR[23]=$SCR_GRP[1].$MCH_POS_X;
:SR[24]=$SCR_GRP[1].$MCH_POS_Y;
2818: L P[2818] 800cm/min CNT100 COORD PTH ;
:SR[23]=$SCR_GRP[1].$MCH_POS_X;
:SR[24]=$SCR_GRP[1].$MCH_POS_Y;
2819: L P[2819] 800cm/min CNT100 COORD PTH ;
:SR[23]=$SCR_GRP[1].$MCH_POS_X;
:SR[24]=$SCR_GRP[1].$MCH_POS_Y;
2820: L P[2820] 800cm/min CNT100 COORD PTH ;
:SR[23]=$SCR_GRP[1].$MCH_POS_X;
:SR[24]=$SCR_GRP[1].$MCH_POS_Y;
2821: L P[2821] 800cm/min CNT100 COORD PTH ;
:SR[23]=$SCR_GRP[1].$MCH_POS_X;
:SR[24]=$SCR_GRP[1].$MCH_POS_Y;
2822: L P[2822] 800cm/min CNT100 COORD PTH ;
:SR[23]=$SCR_GRP[1].$MCH_POS_X;
:SR[24]=$SCR_GRP[1].$MCH_POS_Y;
2823: L P[2823] 800cm/min CNT100 COORD PTH ;
:SR[23]=$SCR_GRP[1].$MCH_POS_X;
:SR[24]=$SCR_GRP[1].$MCH_POS_Y;
2824: L P[2824] 800cm/min CNT100 COORD PTH ;
:SR[23]=$SCR_GRP[1].$MCH_POS_X;
:SR[24]=$SCR_GRP[1].$MCH_POS_Y;
2825: L P[2825] 800cm/min CNT100 COORD PTH ;
:SR[23]=$SCR_GRP[1].$MCH_POS_X;
:SR[24]=$SCR_GRP[1].$MCH_POS_Y;
2826: L P[2826] 800cm/min CNT100 COORD PTH ;
:SR[23]=$SCR_GRP[1].$MCH_POS_X;
:SR[24]=$SCR_GRP[1].$MCH_POS_Y;
2827: L P[2827] 800cm/min CNT100 COORD PTH ;
:SR[23]=$SCR_GRP[1].$MCH_POS_X;
:SR[24]=$SCR_GRP[1].$MCH_POS_Y;
2828: L P[2828] 800cm/min CNT100 COORD PTH ;
:SR[23]=$SCR_GRP[1].$MCH_POS_X;
:SR[24]=$SCR_GRP[1].$MCH_POS_Y;
2829: L P[2829] 800cm/min CNT100 COORD PTH ;
:SR[23]=$SCR_GRP[1].$MCH_POS_X;
:SR[24]=$SCR_GRP[1].$MCH_POS_Y;
2830: L P[2830] 800cm/min CNT100 COORD PTH ;
:SR[23]=$SCR_GRP[1].$MCH_POS_X;
:SR[24]=$SCR_GRP[1].$MCH_POS_Y;
2831: L P[2831] 800cm/min CNT100 COORD PTH ;
:SR[23]=$SCR_GRP[1].$MCH_POS_X;
:SR[24]=$SCR_GRP[1].$MCH_POS_Y;
2832: L P[2832] 800cm/min CNT100 COORD PTH ;
:SR[23]=$SCR_GRP[1].$MCH_POS_X;
:SR[24]=$SCR_GRP[1].$MCH_POS_Y;
2833: L P[2833] 800cm/min CNT100 COORD PTH ;
:SR[23]=$SCR_GRP[1].$MCH_POS_X;
:SR[24]=$SCR_GRP[1].$MCH_POS_Y;
2834: L P[2834] 800cm/min CNT100 COORD PTH ;
:SR[23]=$SCR_GRP[1].$MCH_POS_X;
:SR[24]=$SCR_GRP[1].$MCH_POS_Y;
2835: L P[2835] 800cm/min CNT100 COORD PTH ;
:SR[23]=$SCR_GRP[1].$MCH_POS_X;
:SR[24]=$SCR_GRP[1].$MCH_POS_Y;
2836: L P[2836] 800cm/min CNT100 COORD PTH ;
:SR[23]=$SCR_GRP[1].$MCH_POS_X;
:SR[24]=$SCR_GRP[1].$MCH_POS_Y;
2837: L P[2837] 800cm/min CNT100 COORD PTH ;
:SR[23]=$SCR_GRP[1].$MCH_POS_X;
:SR[24]=$SCR_GRP[1].$MCH_POS_Y;
2838: L P[2838] 800cm/min CNT100 COORD PTH ;
:SR[23]=$SCR_GRP[1].$MCH_POS_X;
:SR[24]=$SCR_GRP[1].$MCH_POS_Y;
2839: L P[2839] 800cm/min CNT100 COORD PTH ;
:SR[23]=$SCR_GRP[1].$MCH_POS_X;
:SR[24]=$SCR_GRP[1].$MCH_POS_Y;
2840: L P[2840] 800cm/min CNT100 COORD PTH ;
:SR[23]=$SCR_GRP[1].$MCH_POS_X;
:SR[24]=$SCR_GRP[1].$MCH_POS_Y;
2841: L P[2841] 800cm/min CNT100 COORD PTH ;
:SR[23]=$SCR_GRP[1].$MCH_POS_X;
:SR[24]=$SCR_GRP[1].$MCH_POS_Y;
2842: L P[2842] 800cm/min CNT100 COORD PTH ;
:SR[23]=$SCR_GRP[1].$MCH_POS_X;
:SR[24]=$SCR_GRP[1].$MCH_POS_Y;
2843: L P[2843] 800cm/min CNT100 COORD PTH ;
:SR[23]=$SCR_GRP[1].$MCH_POS_X;
:SR[24]=$SCR_GRP[1].$MCH_POS_Y;
2844: L P[2844] 800cm/min CNT100 COORD PTH ;
:SR[23]=$SCR_GRP[1].$MCH_POS_X;
:SR[24]=$SCR_GRP[1].$MCH_POS_Y;
2845: L P[2845] 800cm/min CNT100 COORD PTH ;
:SR[23]=$SCR_GRP[1].$MCH_POS_X;
:SR[24]=$SCR_GRP[1].$MCH_POS_Y;
2846: L P[2846] 800cm/min CNT100 COORD PTH ;
:SR[23]=$SCR_GRP[1].$MCH_POS_X;
:SR[24]=$SCR_GRP[1].$MCH_POS_Y;
2847: L P[2847] 800cm/min CNT100 COORD PTH ;
:SR[23]=$SCR_GRP[1].$MCH_POS_X;
:SR[24]=$SCR_GRP[1].$MCH_POS_Y;
2848: L P[2848] 800cm/min CNT100 COORD PTH ;
:SR[23]=$SCR_GRP[1].$MCH_POS_X;
:SR[24]=$SCR_GRP[1].$MCH_POS_Y;
2849: L P[2849] 800cm/min CNT100 COORD PTH ;
:SR[23]=$SCR_GRP[1].$MCH_POS_X;
:SR[24]=$SCR_GRP[1].$MCH_POS_Y;
2850: L P[2850] 800cm/min CNT100 COORD PTH ;
:SR[23]=$SCR_GRP[1].$MCH_POS_X;
:SR[24]=$SCR_GRP[1].$MCH_POS_Y;
2851: L P[2851] 800cm/min CNT100 COORD PTH ;
:SR[23]=$SCR_GRP[1].$MCH_POS_X;
:SR[24]=$SCR_GRP[1].$MCH_POS_Y;
2852: L P[2852] 800cm/min CNT100 COORD PTH ;
:SR[23]=$SCR_GRP[1].$MCH_POS_X;
:SR[24]=$SCR_GRP[1].$MCH_POS_Y;
2853: L P[2853] 800cm/min CNT100 COORD PTH ;
:SR[23]=$SCR_GRP[1].$MCH_POS_X;
:SR[24]=$SCR_GRP[1].$MCH_POS_Y;
2854: L P[2854] 800cm/min CNT100 COORD PTH ;
:SR[23]=$SCR_GRP[1].$MCH_POS_X;
:SR[24]=$SCR_GRP[1].$MCH_POS_Y;
2855: L P[2855] 800cm/min CNT100 COORD PTH ;
:SR[23]=$SCR_GRP[1].$MCH_POS_X;
:SR[24]=$SCR_GRP[1].$MCH_POS_Y;
2856: L P[2856] 800cm/min CNT100 COORD PTH ;
:SR[23]=$SCR_GRP[1].$MCH_POS_X;
:SR[24]=$SCR_GRP[1].$MCH_POS_Y;
2857: L P[2857] 800cm/min CNT100 COORD PTH ;
:SR[23]=$SCR_GRP[1].$MCH_POS_X;
:SR[24]=$SCR_GRP[1].$MCH_POS_Y;
2858: L P[2858] 800cm/min CNT100 COORD PTH ;
:SR[23]=$SCR_GRP[1].$MCH_POS_X;
:SR[24]=$SCR_GRP[1].$MCH_POS_Y;
2859: L P[2859] 800cm/min CNT100 COORD PTH ;
:SR[23]=$SCR_GRP[1].$MCH_POS_X;
:SR[24]=$SCR_GRP[1].$MCH_POS_Y;
2860: L P[2860] 800cm/min CNT100 COORD PTH ;
:SR[23]=$SCR_GRP[1].$MCH_POS_X;
:SR[24]=$SCR_GRP[1].$MCH_POS_Y;
2861: L P[2861] 800cm/min CNT100 COORD PTH ;
:SR[23]=$SCR_GRP[1].$MCH_POS_X;
:SR[24]=$SCR_GRP[1].$MCH_POS_Y;
2862: L P[2862] 800cm/min CNT100 COORD PTH ;
:SR[23]=$SCR_GRP[1].$MCH_POS_X;
:SR[24]=$SCR_GRP[1].$MCH_POS_Y;
2863: L P[2863] 800cm/min CNT100 COORD PTH ;
:SR[23]=$SCR_GRP[1].$MCH_POS_X;
:SR[24]=$SCR_GRP[1].$MCH_POS_Y;
2864: L P[2864] 800cm/min CNT100 COORD PTH ;
:SR[23]=$SCR_GRP[1].$MCH_POS_X;
:SR[24]=$SCR_GRP[1].$MCH_POS_Y;
2865: L P[2865] 800cm/min CNT100 COORD PTH ;
:SR[23]=$SCR_GRP[1].$MCH_POS_X;
:SR[24]=$SCR_GRP[1].$MCH_POS_Y;
2866: L P[2866] 800cm/min CNT100 COORD PTH ;
:SR[23]=$SCR_GRP[1].$MCH_POS_X;
:SR[24]=$SCR_GRP[1].$MCH_POS_Y;
2867: L P[2867] 800cm/min CNT100 COORD PTH ;
:SR[23]=$SCR_GRP[1].$MCH_POS_X;
:SR[24]=$SCR_GRP[1].$MCH_POS_Y;
2868: L P[2868] 800cm/min CNT100 COORD PTH ;
:SR[23]=$SCR_GRP[1].$MCH_POS_X;
:SR[24]=$SCR_GRP[1].$MCH_POS_Y;
2869: L P[2869] 800cm/min CNT100 COORD PTH ;
:SR[23]=$SCR_GRP[1].$MCH_POS_X;
:SR[24]=$SCR_GRP[1].$MCH_POS_Y;
2870: L P[2870] 800cm/min CNT100 COORD PTH ;
:SR[23]=$SCR_GRP[1].$MCH_POS_X;
:SR[24]=$SCR_GRP[1].$MCH_POS_Y;
2871: L P[2871] 800cm/min CNT100 COORD PTH ;
:SR[23]=$SCR_GRP[1].$MCH_POS_X;
:SR[24]=$SCR_GRP[1].$MCH_POS_Y;
2872: L P[2872] 800cm/min CNT100 COORD PTH ;
:SR[23]=$SCR_GRP[1].$MCH_POS_X;
:SR[24]=$SCR_GRP[1].$MCH_POS_Y;
2873: L P[2873] 800cm/min CNT100 COORD PTH ;
:SR[23]=$SCR_GRP[1].$MCH_POS_X;
:SR[24]=$SCR_GRP[1].$MCH_POS_Y;
2874: L P[2874] 800cm/min CNT100 COORD PTH ;
:SR[23]=$SCR_GRP[1].$MCH_POS_X;
:SR[24]=$SCR_GRP[1].$MCH_POS_Y;
2875: L P[2875] 800cm/min CNT100 COORD PTH ;
:SR[23]=$SCR_GRP[1].$MCH_POS_X;
:SR[24]=$SCR_GRP[1].$MCH_POS_Y;
2876: L P[2876] 800cm/min CNT100 COORD PTH ;
:SR[23]=$SCR_GRP[1].$MCH_POS_X;
:SR[24]=$SCR_GRP[1].$MCH_POS_Y;
2877: L P[2877] 800cm/min CNT100 COORD PTH ;
:SR[23]=$SCR_GRP[1].$MCH_POS_X;
:SR[24]=$SCR_GRP[1].$MCH_POS_Y;
2878: L P[2878] 800cm/min CNT100 COORD PTH ;
:SR[23]=$SCR_GRP[1].$MCH_POS_X;
:SR[24]=$SCR_GRP[1].$MCH_POS_Y;
2879: L P[2879] 800cm/min CNT100 COORD PTH ;
:SR[23]=$SCR_GRP[1].$MCH_POS_X;
:SR[24]=$SCR_GRP[1].$MCH_POS_Y;
2880: L P[2880] 800cm/min CNT100 COORD PTH ;
:SR[23]=$SCR_GRP[1].$MCH_POS_X;
:SR[24]=$SCR_GRP[1].$MCH_POS_Y;
2881: L P[2881] 800cm/min CNT100 COORD PTH ;
:SR[23]=$SCR_GRP[1].$MCH_POS_X;
:SR[24]=$SCR_GRP[1].$MCH_POS_Y;
2882: L P[2882] 800cm/min CNT100 COORD PTH ;
:SR[23]=$SCR_GRP[1].$MCH_POS_X;
:SR[24]=$SCR_GRP[1].$MCH_POS_Y;
2883: L P[2883] 800cm/min CNT100 COORD PTH ;
:SR[23]=$SCR_GRP[1].$MCH_POS_X;
:SR[24]=$SCR_GRP[1].$MCH_POS_Y;
2884: L P[2884] 800cm/min CNT100 COORD PTH ;
:SR[23]=$SCR_GRP[1].$MCH_POS_X;
:SR[24]=$SCR_GRP[1].$MCH_POS_Y;
2885: L P[2885] 800cm/min CNT100 COORD PTH ;
:SR[23]=$SCR_GRP[1].$MCH_POS_X;
:SR[24]=$SCR_GRP[1].$MCH_POS_Y;
2886: L P[2886] 800cm/min CNT100 COORD PTH ;
:SR[23]=$SCR_GRP[1].$MCH_POS_X;
:SR[24]=$SCR_GRP[1].$MCH_POS_Y;
2887: L P[2887] 800cm/min CNT100 COORD PTH ;
:SR[23]=$SCR_GRP[1].$MCH_POS_X;
:SR[24]=$SCR_GRP[1].$MCH_POS_Y;
2888: L P[2888] 800cm/min CNT100 COORD PTH ;
:SR[23]=$SCR_GRP[1].$MCH_POS_X;
:SR[24]=$SCR_GRP[1].$MCH_POS_Y;
2889: L P[2889] 800cm/min CNT100 COORD PTH ;
:SR[23]=$SCR_GRP[1].$MCH_POS_X;
:SR[24]=$SCR_GRP[1].$MCH_POS_Y;
2890: L P[2890] 800cm/min CNT100 COORD PTH ;
:SR[23]=$SCR_GRP[1].$MCH_POS_X;
:SR[24]=$SCR_GRP[1].$MCH_POS_Y;
2891: L P[2891] 800cm/min CNT100 COORD PTH ;
:SR[23]=$SCR_GRP[1].$MCH_POS_X;
:SR[24]=$SCR_GRP[1].$MCH_POS_Y;
2892: L P[2892] 800cm/min CNT100 COORD PTH ;
:SR[23]=$SCR_GRP[1].$MCH_POS_X;
:SR[24]=$SCR_GRP[1].$MCH_POS_Y;
2893: L P[2893] 800cm/min CNT100 COORD PTH ;
:SR[23]=$SCR_GRP[1].$MCH_POS_X;
:SR[24]=$SCR_GRP[1].$MCH_POS_Y;
2894: L P[2894] 800cm/min CNT100 COORD PTH ;
:SR[23]=$SCR_GRP[1].$MCH_POS_X;
:SR[24]=$SCR_GRP[1].$MCH_POS_Y;
2895: L P[2895] 800cm/min CNT100 COORD PTH ;
:SR[23]=$SCR_GRP[1].$MCH_POS_X;
:SR[24]=$SCR_GRP[1].$MCH_POS_Y;
2896: L P[2896] 800cm/min CNT100 COORD PTH ;
:SR[23]=$SCR_GRP[1].$MCH_POS_X;
:SR[24]=$SCR_GRP[1].$MCH_POS_Y;
2897: L P[2897] 800cm/min CNT100 COORD PTH ;
:SR[23]=$SCR_GRP[1].$MCH_POS_X;
:SR[24]=$SCR_GRP[1].$MCH_POS_Y;
2898: L P[2898] 800cm/min CNT100 COORD PTH ;
:SR[23]=$SCR_GRP[1].$MCH_POS_X;
:SR[24]=$SCR_GRP[1].$MCH_POS_Y;
2899: L P[2899] 800cm/min CNT100 COORD PTH ;
:SR[23]=$SCR_GRP[1].$MCH_POS_X;
:SR[24]=$SCR_GRP[1].$MCH_POS_Y;
2900: L P[2900] 800cm/min CNT100 COORD PTH ;
:SR[23]=$SCR_GRP[1].$MCH_POS_X;
:SR[24]=$SCR_GRP[1].$MCH_POS_Y;
2901: L P[2901] 800cm/min CNT100 COORD PTH ;
:SR[23]=$SCR_GRP[1].$MCH_POS_X;
:SR[24]=$SCR_GRP[1].$MCH_POS_Y;
2902: L P[2902] 800cm/min CNT100 COORD PTH ;
:SR[23]=$SCR_GRP[1].$MCH_POS_X;
:SR[24]=$SCR_GRP[1].$MCH_POS_Y;
2903: L P[2903] 800cm/min CNT100 COORD PTH ;
:SR[23]=$SCR_GRP[1].$MCH_POS_X;
:SR[24]=$SCR_GRP[1].$MCH_POS_Y;
2904: L P[2904] 800cm/min CNT100 COORD PTH ;
:SR[23]=$SCR_GRP[1].$MCH_POS_X;
:SR[24]=$SCR_GRP[1].$MCH_POS_Y;
2905: L P[2905] 800cm/min CNT100 COORD PTH ;
:SR[23]=$SCR_GRP[1].$MCH_POS_X;
:SR[24]=$SCR_GRP[1].$MCH_POS_Y;
2906: L P[2906] 800cm/min CNT100 COORD PTH ;
:SR[23]=$SCR_GRP[1].$MCH_POS_X;
:SR[24]=$SCR_GRP[1].$MCH_POS_Y;
2907: L P[2907] 800cm/min CNT100 COORD PTH ;
:SR[23]=$SCR_GRP[1].$MCH_POS_X;
:SR[24]=$SCR_GRP[1].$MCH_POS_Y;
2908: L P[2908] 800cm/min CNT100 COORD PTH ;
:SR[23]=$SCR_GRP[1].$MCH_POS_X;
:SR[24]=$SCR_GRP[1].$MCH_POS_Y;
2909: L P[2909] 800cm/min CNT100 COORD PTH ;
:SR[23]=$SCR_GRP[1].$MCH_POS_X;
:SR[24]=$SCR_GRP[1].$MCH_POS_Y;
2910: L P[2910] 800cm/min CNT100 COORD PTH ;
:SR[23]=$SCR_GRP[1].$MCH_POS_X;
:SR[24]=$SCR_GRP[1].$MCH_POS_Y;
2911: L P[2911] 800cm/min CNT100 COORD PTH ;
:SR[23]=$SCR_GRP[1].$MCH_POS_X;
:SR[24]=$SCR_GRP[1].$MCH_POS_Y;
2912: L P[2912] 800cm/min CNT100 COORD PTH ;
:SR[23]=$SCR_GRP[1].$MCH_POS_X;
:SR[24]=$SCR_GRP[1].$MCH_POS_Y;
2913: L P[2913] 800cm/min CNT100 COORD PTH ;
:SR[23]=$SCR_GRP[1].$MCH_POS_X;
:SR[24]=$SCR_GRP[1].$MCH_POS_Y;
2914: L P[2914] 800cm/min CNT100 COORD PTH ;
:SR[23]=$SCR_GRP[1].$MCH_POS_X;
:SR[24]=$SCR_GRP[1].$MCH_POS_Y;
2915: L P[2915] 800cm/min CNT100 COORD PTH ;
:SR[23]=$SCR_GRP[1].$MCH_POS_X;
:SR[24]=$SCR_GRP[1].$MCH_POS_Y;
2916: L P[2916] 800cm/min CNT100 COORD PTH ;
:SR[23]=$SCR_GRP[1].$MCH_POS_X;
:SR[24]=$SCR_GRP[1].$MCH_POS_Y;
2917: L P[2917] 800cm/min CNT100 COORD PTH ;
:SR[23]=$SCR_GRP[1].$MCH_POS_X;
:SR[24]=$SCR_GRP[1].$MCH_POS_Y;
2918: L P[2918] 800cm/min CNT100 COORD PTH ;
:SR[23]=$SCR_GRP[1].$MCH_POS_X;
:SR[24]=$SCR_GRP[1].$MCH_POS_Y;
2919: L P[2919] 800cm/min CNT100 COORD PTH ;
:SR[23]=$SCR_GRP[1].$MCH_POS_X;
:SR[24]=$SCR_GRP[1].$MCH_POS_Y;
2920: L P[2920] 800cm/min CNT100 COORD PTH ;
:SR[23]=$SCR_GRP[1].$MCH_POS_X;
:SR[24]=$SCR_GRP[1].$MCH_POS_Y;
2921: L P[2921] 800cm/min CNT100 COORD PTH ;
:SR[23]=$SCR_GRP[1].$MCH_POS_X;
:SR[24]=$SCR_GRP[1].$MCH_POS_Y;
2922: L P[2922] 800cm/min CNT100 COORD PTH ;
:SR[23]=$SCR_GRP[1].$MCH_POS_X;
:SR[24]=$SCR_GRP[1].$MCH_POS_Y;
2923: L P[2923] 800cm/min CNT100 COORD PTH ;
:SR[23]=$SCR_GRP[1].$MCH_POS_X;
:SR[24]=$SCR_GRP[1].$MCH_POS_Y;
2924: L P[2924] 800cm/min CNT100 COORD PTH ;
:SR[23]=$SCR_GRP[1].$MCH_POS_X;
:SR[24]=$SCR_GRP[1].$MCH_POS_Y;
2925: L P[2925] 800cm/min CNT100 COORD PTH ;
:SR[23]=$SCR_GRP[1].$MCH_POS_X;
:SR[24]=$SCR_GRP[1].$MCH_POS_Y;
2926: L P[2926] 800cm/min CNT100 COORD PTH ;
:SR[23]=$SCR_GRP[1].$MCH_POS_X;
:SR[24]=$SCR_GRP[1].$MCH_POS_Y;
2927: L P[2927] 800cm/min CNT100 COORD PTH ;
:SR[23]=$SCR_GRP[1].$MCH_POS_X;
:SR[24]=$SCR_GRP[1].$MCH_POS_Y;
2928: L P[2928] 800cm/min CNT100 COORD PTH ;
:SR[23]=$SCR_GRP[1].$MCH_POS_X;
:SR[24]=$SCR_GRP[1].$MCH_POS_Y;
2929: L P[2929] 800cm/min CNT100 COORD PTH ;
:SR[23]=$SCR_GRP[1].$MCH_POS_X;
:SR[24]=$SCR_GRP[1].$MCH_POS_Y;
2930: L P[2930] 800cm/min CNT100 COORD PTH ;
:SR[23]=$SCR_GRP[1].$MCH_POS_X;
:SR[24]=$SCR_GRP[1].$MCH_POS_Y;
2931: L P[2931] 800cm/min CNT100 COORD PTH ;
:SR[23]=$SCR_GRP[1].$MCH_POS_X;
:SR[24]=$SCR_GRP[1].$MCH_POS_Y;
2932: L P[2932] 800cm/min CNT100 COORD PTH ;
:SR[23]=$SCR_GRP[1].$MCH_POS_X;
:SR[24]=$SCR_GRP[1].$MCH_POS_Y;
2933: L P[2933] 800cm/min CNT100 COORD PTH ;
:SR[23]=$SCR_GRP[1].$MCH_POS_X;
:SR[24]=$SCR_GRP[1].$MCH_POS_Y;
2934: L P[2934] 800cm/min CNT100 COORD PTH ;
:SR[23]=$SCR_GRP[1].$MCH_POS_X;
:SR[24]=$SCR_GRP[1].$MCH_POS_Y;
2935: L P[2935] 800cm/min CNT100 COORD PTH ;
:SR[23]=$SCR_GRP[1].$MCH_POS_X;
:SR[24]=$SCR_GRP[1].$MCH_POS_Y;
2936: L P[2936] 800cm/min CNT100 COORD PTH ;
:SR[23]=$SCR_GRP[1].$MCH_POS_X;
:SR[24]=$SCR_GRP[1].$MCH_POS_Y;
2937: L P[2937] 800cm/min CNT100 COORD PTH ;
:SR[23]=$SCR_GRP[1].$MCH_POS_X;
:SR[24]=$SCR_GRP[1].$MCH_POS_Y;
2938: L P[2938] 800cm/min CNT100 COORD PTH ;
:SR[23]=$SCR_GRP[1].$MCH_POS_X;
:SR[24]=$SCR_GRP[1].$MCH_POS_Y;
2939: L P[2939] 800cm/min CNT100 COORD PTH ;
:SR[23]=$SCR_GRP[1].$MCH_POS_X;
:SR[24]=$SCR_GRP[1].$MCH_POS_Y;
2940: L P[2940] 800cm/min CNT100 COORD PTH ;
:SR[23]=$SCR_GRP[1].$MCH_POS_X;
:SR[24]=$SCR_GRP[1].$MCH_POS_Y;
2941: L P[2941] 800cm/min CNT100 COORD PTH ;
:SR[23]=$SCR_GRP[1].$MCH_POS_X;
:SR[24]=$SCR_GRP[1].$MCH_POS_Y;
2942: L P[2942] 800cm/min CNT100 COORD PTH ;
:SR[23]=$SCR_GRP[1].$MCH_POS_X;
:SR[24]=$SCR_GRP[1].$MCH_POS_Y;
2943: L P[2943] 800cm/min CNT100 COORD PTH ;
:SR[23]=$SCR_GRP[1].$MCH_POS_X;
